SYSTEM temexdmod
  (* Version 1.0, Author, 4DIAC-Consortium *)
  APPLICATION looptest
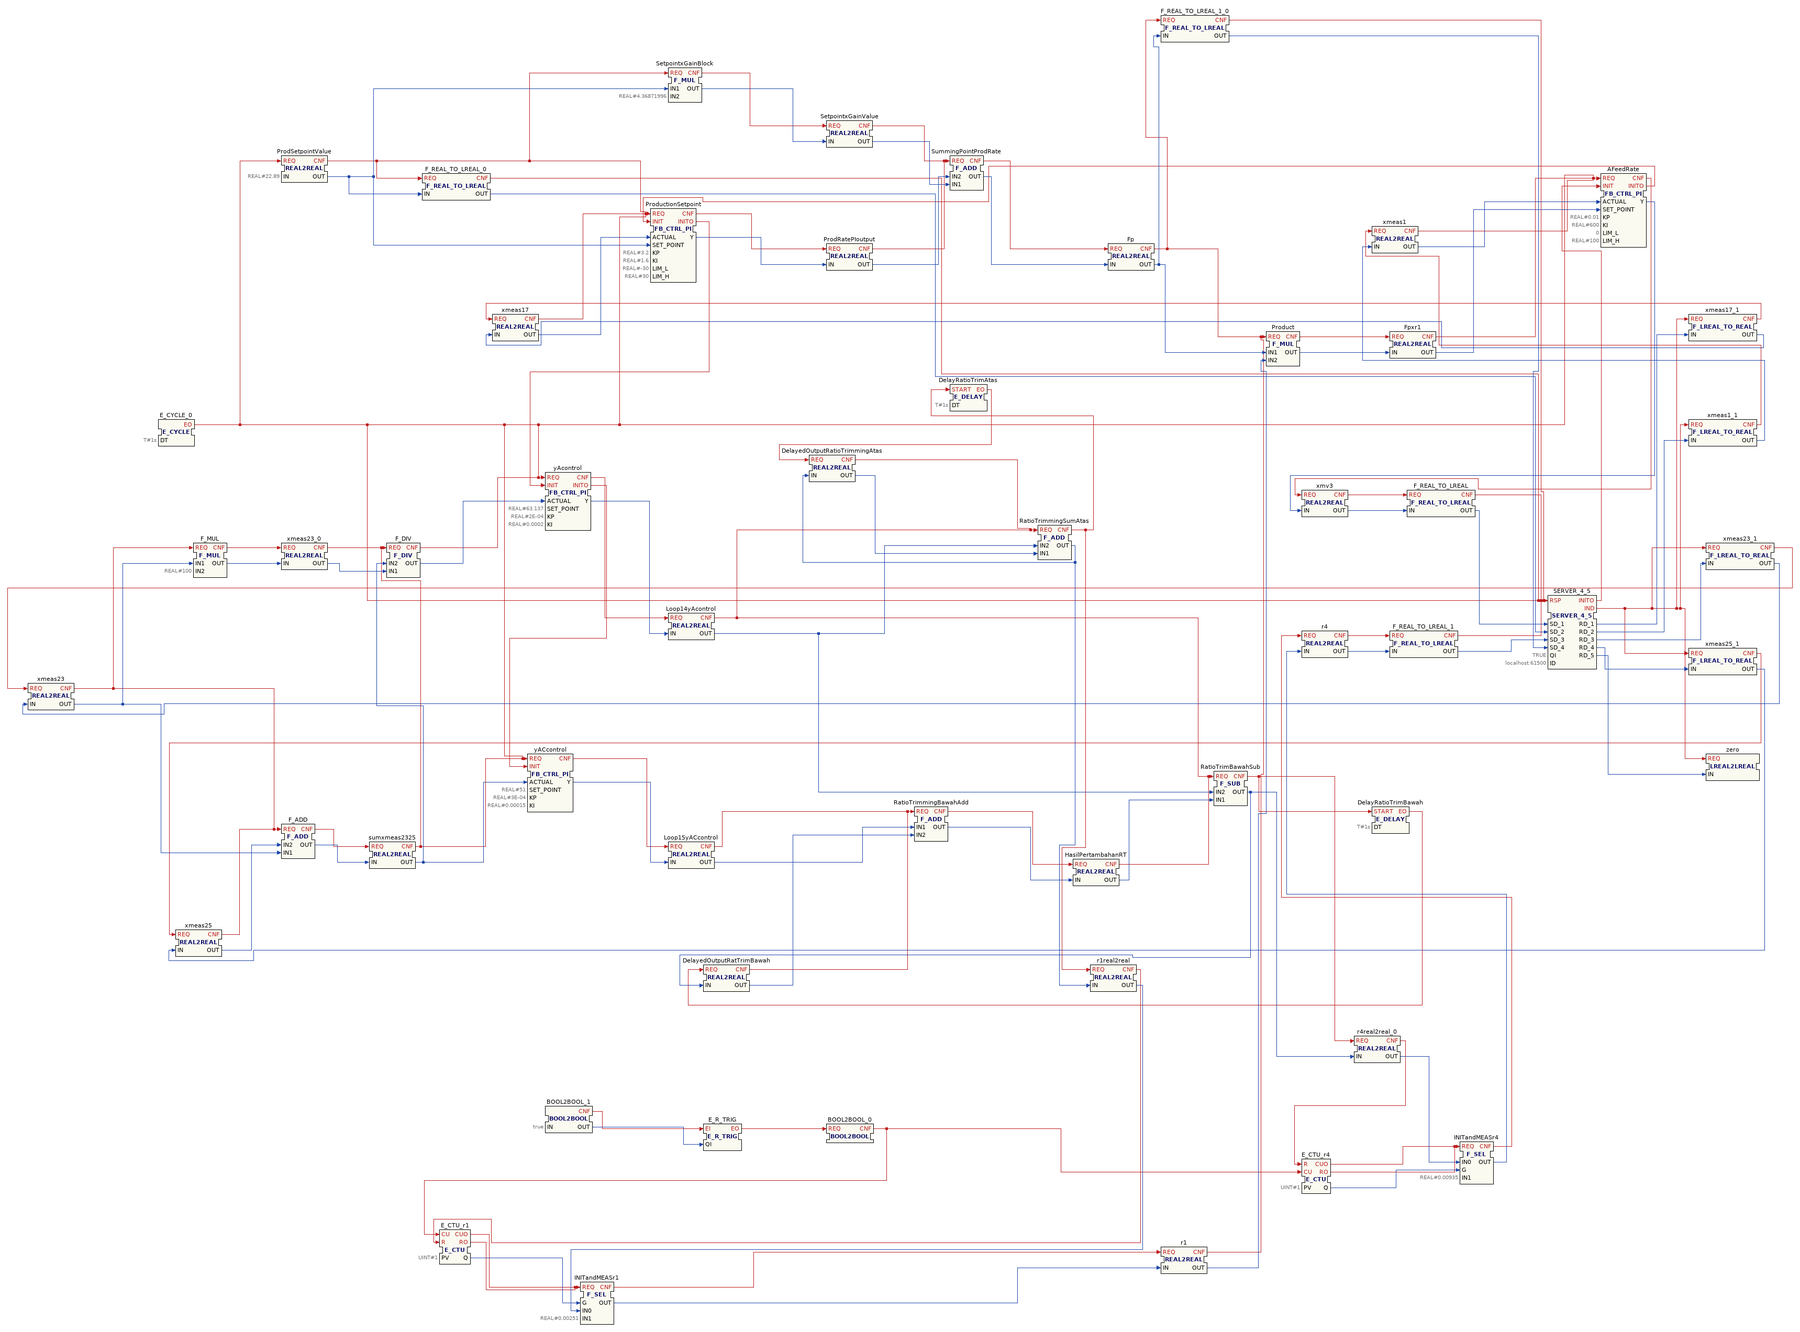
    FBS
      AFeedRate : FB_CTRL_PI(KP := REAL#0.01, KI := REAL#600, LIM_L := 0, LIM_H := REAL#100);
      ProductionSetpoint : FB_CTRL_PI(KP := REAL#3.2, KI := REAL#1.6, LIM_L := REAL#-30, LIM_H := REAL#30);
      Product : F_MUL;
      xmeas1 : REAL2REAL;
      Fpxr1 : REAL2REAL;
      xmv3 : REAL2REAL;
      SummingPointProdRate : F_ADD;
      ProdRatePIoutput : REAL2REAL;
      Fp : REAL2REAL;
      SetpointxGainBlock : F_MUL(IN2 := REAL#4.36871996);
      SetpointxGainValue : REAL2REAL;
      yAcontrol : FB_CTRL_PI(SET_POINT := REAL#63.137, KP := REAL#2E-04, KI := REAL#0.0002);
      yACcontrol : FB_CTRL_PI(SET_POINT := REAL#51, KP := REAL#3E-04, KI := REAL#0.00015);
      Loop14yAcontrol : REAL2REAL;
      Loop15yACcontrol : REAL2REAL;
      RatioTrimBawahSub : F_SUB;
      RatioTrimmingBawahAdd : F_ADD;
      HasilPertambahanRT : REAL2REAL;
      DelayRatioTrimBawah : E_DELAY(DT := T#1s);
      DelayedOutputRatTrimBawah : REAL2REAL;
      r4 : REAL2REAL;
      RatioTrimmingSumAtas : F_ADD;
      DelayedOutputRatioTrimmingAtas : REAL2REAL;
      DelayRatioTrimAtas : E_DELAY(DT := T#1s);
      xmeas17 : REAL2REAL;
      xmeas25 : REAL2REAL;
      F_ADD : F_ADD;
      sumxmeas2325 : REAL2REAL;
      F_MUL : F_MUL(IN2 := REAL#100);
      F_DIV : F_DIV;
      BOOL2BOOL_0 : BOOL2BOOL;
      E_CTU_r1 : E_CTU(PV := UINT#1);
      E_CYCLE_0 : E_CYCLE(DT := T#1s);
      r1real2real : REAL2REAL;
      BOOL2BOOL_1 : BOOL2BOOL(IN := true);
      INITandMEASr1 : F_SEL(IN1 := REAL#0.00251);
      E_R_TRIG : E_R_TRIG;
      r1 : REAL2REAL;
      SERVER_4_5 : SERVER_4_5(QI := TRUE, ID := localhost:61500);
      E_CTU_r4 : E_CTU(PV := UINT#1);
      INITandMEASr4 : F_SEL(IN1 := REAL#0.00935);
      r4real2real_0 : REAL2REAL;
      ProdSetpointValue : REAL2REAL(IN := REAL#22.89);
      F_REAL_TO_LREAL : F_REAL_TO_LREAL;
      F_REAL_TO_LREAL_0 : F_REAL_TO_LREAL;
      F_REAL_TO_LREAL_1 : F_REAL_TO_LREAL;
      F_REAL_TO_LREAL_1_0 : F_REAL_TO_LREAL;
      xmeas17_1 : F_LREAL_TO_REAL;
      xmeas1_1 : F_LREAL_TO_REAL;
      xmeas23_1 : F_LREAL_TO_REAL;
      xmeas25_1 : F_LREAL_TO_REAL;
      xmeas23 : REAL2REAL;
      xmeas23_0 : REAL2REAL;
      zero : LREAL2LREAL;
    END_FBS
    EVENT_CONNECTIONS
      Loop15yACcontrol.CNF TO RatioTrimmingBawahAdd.REQ;
      RatioTrimBawahSub.CNF TO DelayRatioTrimBawah.START;
      DelayRatioTrimBawah.EO TO DelayedOutputRatTrimBawah.REQ;
      DelayedOutputRatTrimBawah.CNF TO RatioTrimmingBawahAdd.REQ;
      Loop14yAcontrol.CNF TO RatioTrimmingSumAtas.REQ;
      Fp.CNF TO Product.REQ;
      RatioTrimmingSumAtas.CNF TO DelayRatioTrimAtas.START;
      DelayRatioTrimAtas.EO TO DelayedOutputRatioTrimmingAtas.REQ;
      DelayedOutputRatioTrimmingAtas.CNF TO RatioTrimmingSumAtas.REQ;
      SummingPointProdRate.CNF TO Fp.REQ;
      xmeas17.CNF TO ProductionSetpoint.REQ;
      SetpointxGainBlock.CNF TO SetpointxGainValue.REQ;
      SetpointxGainValue.CNF TO SummingPointProdRate.REQ;
      ProductionSetpoint.CNF TO ProdRatePIoutput.REQ;
      ProdRatePIoutput.CNF TO SummingPointProdRate.REQ;
      F_ADD.CNF TO sumxmeas2325.REQ;
      xmeas25.CNF TO F_ADD.REQ;
      sumxmeas2325.CNF TO yACcontrol.REQ;
      yACcontrol.CNF TO Loop15yACcontrol.REQ;
      F_DIV.CNF TO yAcontrol.REQ;
      yAcontrol.CNF TO Loop14yAcontrol.REQ;
      RatioTrimmingBawahAdd.CNF TO HasilPertambahanRT.REQ;
      HasilPertambahanRT.CNF TO RatioTrimBawahSub.REQ;
      Loop14yAcontrol.CNF TO RatioTrimBawahSub.REQ;
      Product.CNF TO Fpxr1.REQ;
      Fpxr1.CNF TO AFeedRate.REQ;
      xmeas1.CNF TO AFeedRate.REQ;
      AFeedRate.CNF TO xmv3.REQ;
      BOOL2BOOL_1.CNF TO E_R_TRIG.EI;
      E_R_TRIG.EO TO BOOL2BOOL_0.REQ;
      E_CTU_r1.CUO TO INITandMEASr1.REQ;
      E_CTU_r1.RO TO INITandMEASr1.REQ;
      BOOL2BOOL_0.CNF TO E_CTU_r1.CU;
      r1.CNF TO Product.REQ;
      RatioTrimmingSumAtas.CNF TO r1real2real.REQ;
      r1real2real.CNF TO E_CTU_r1.R;
      INITandMEASr1.CNF TO r1.REQ;
      AFeedRate.INITO TO ProductionSetpoint.INIT;
      ProductionSetpoint.INITO TO yAcontrol.INIT;
      yAcontrol.INITO TO yACcontrol.INIT;
      E_CYCLE_0.EO TO ProductionSetpoint.REQ;
      E_CYCLE_0.EO TO yAcontrol.REQ;
      E_CYCLE_0.EO TO yACcontrol.REQ;
      E_CYCLE_0.EO TO AFeedRate.REQ;
      SERVER_4_5.INITO TO AFeedRate.INIT;
      E_CYCLE_0.EO TO SERVER_4_5.RSP;
      INITandMEASr4.CNF TO r4.REQ;
      r4real2real_0.CNF TO E_CTU_r4.R;
      RatioTrimBawahSub.CNF TO r4real2real_0.REQ;
      BOOL2BOOL_0.CNF TO E_CTU_r4.CU;
      E_CTU_r4.CUO TO INITandMEASr4.REQ;
      E_CTU_r4.RO TO INITandMEASr4.REQ;
      E_CYCLE_0.EO TO ProdSetpointValue.REQ;
      ProdSetpointValue.CNF TO SetpointxGainBlock.REQ;
      ProdSetpointValue.CNF TO ProductionSetpoint.REQ;
      xmv3.CNF TO F_REAL_TO_LREAL.REQ;
      F_REAL_TO_LREAL.CNF TO SERVER_4_5.RSP;
      ProdSetpointValue.CNF TO F_REAL_TO_LREAL_0.REQ;
      F_REAL_TO_LREAL_0.CNF TO SERVER_4_5.RSP;
      r4.CNF TO F_REAL_TO_LREAL_1.REQ;
      F_REAL_TO_LREAL_1.CNF TO SERVER_4_5.RSP;
      F_REAL_TO_LREAL_1_0.CNF TO SERVER_4_5.RSP;
      Fp.CNF TO F_REAL_TO_LREAL_1_0.REQ;
      xmeas17_1.CNF TO xmeas17.REQ;
      SERVER_4_5.IND TO xmeas17_1.REQ;
      SERVER_4_5.IND TO xmeas1_1.REQ;
      xmeas1_1.CNF TO xmeas1.REQ;
      SERVER_4_5.IND TO xmeas23_1.REQ;
      xmeas23.CNF TO F_MUL.REQ;
      xmeas23.CNF TO F_ADD.REQ;
      xmeas23_1.CNF TO xmeas23.REQ;
      xmeas25_1.CNF TO xmeas25.REQ;
      SERVER_4_5.IND TO xmeas25_1.REQ;
      xmeas23_0.CNF TO F_DIV.REQ;
      F_MUL.CNF TO xmeas23_0.REQ;
      sumxmeas2325.CNF TO F_DIV.REQ;
      SERVER_4_5.IND TO zero.REQ;
    END_CONNECTIONS
    DATA_CONNECTIONS
      xmeas1.OUT TO AFeedRate.ACTUAL;
      Product.OUT TO Fpxr1.IN;
      Fpxr1.OUT TO AFeedRate.SET_POINT;
      AFeedRate.Y TO xmv3.IN;
      ProductionSetpoint.Y TO ProdRatePIoutput.IN;
      ProdRatePIoutput.OUT TO SummingPointProdRate.IN2;
      SummingPointProdRate.OUT TO Fp.IN;
      Fp.OUT TO Product.IN1;
      SetpointxGainBlock.OUT TO SetpointxGainValue.IN;
      SetpointxGainValue.OUT TO SummingPointProdRate.IN1;
      yAcontrol.Y TO Loop14yAcontrol.IN;
      yACcontrol.Y TO Loop15yACcontrol.IN;
      Loop14yAcontrol.OUT TO RatioTrimBawahSub.IN2;
      Loop15yACcontrol.OUT TO RatioTrimmingBawahAdd.IN1;
      RatioTrimmingBawahAdd.OUT TO HasilPertambahanRT.IN;
      HasilPertambahanRT.OUT TO RatioTrimBawahSub.IN1;
      RatioTrimBawahSub.OUT TO DelayedOutputRatTrimBawah.IN;
      DelayedOutputRatTrimBawah.OUT TO RatioTrimmingBawahAdd.IN2;
      Loop14yAcontrol.OUT TO RatioTrimmingSumAtas.IN2;
      RatioTrimmingSumAtas.OUT TO DelayedOutputRatioTrimmingAtas.IN;
      DelayedOutputRatioTrimmingAtas.OUT TO RatioTrimmingSumAtas.IN1;
      xmeas17.OUT TO ProductionSetpoint.ACTUAL;
      xmeas25.OUT TO F_ADD.IN2;
      F_ADD.OUT TO sumxmeas2325.IN;
      sumxmeas2325.OUT TO yACcontrol.ACTUAL;
      sumxmeas2325.OUT TO F_DIV.IN2;
      F_DIV.OUT TO yAcontrol.ACTUAL;
      E_CTU_r1.Q TO INITandMEASr1.G;
      BOOL2BOOL_1.OUT TO E_R_TRIG.QI;
      RatioTrimmingSumAtas.OUT TO r1real2real.IN;
      r1real2real.OUT TO INITandMEASr1.IN0;
      INITandMEASr1.OUT TO r1.IN;
      r1.OUT TO Product.IN2;
      INITandMEASr4.OUT TO r4.IN;
      RatioTrimBawahSub.OUT TO r4real2real_0.IN;
      r4real2real_0.OUT TO INITandMEASr4.IN0;
      E_CTU_r4.Q TO INITandMEASr4.G;
      ProdSetpointValue.OUT TO ProductionSetpoint.SET_POINT;
      ProdSetpointValue.OUT TO SetpointxGainBlock.IN1;
      xmv3.OUT TO F_REAL_TO_LREAL.IN;
      F_REAL_TO_LREAL.OUT TO SERVER_4_5.SD_1;
      ProdSetpointValue.OUT TO F_REAL_TO_LREAL_0.IN;
      F_REAL_TO_LREAL_0.OUT TO SERVER_4_5.SD_2;
      r4.OUT TO F_REAL_TO_LREAL_1.IN;
      F_REAL_TO_LREAL_1.OUT TO SERVER_4_5.SD_3;
      Fp.OUT TO F_REAL_TO_LREAL_1_0.IN;
      F_REAL_TO_LREAL_1_0.OUT TO SERVER_4_5.SD_4;
      xmeas17_1.OUT TO xmeas17.IN;
      SERVER_4_5.RD_1 TO xmeas17_1.IN;
      xmeas1_1.OUT TO xmeas1.IN;
      SERVER_4_5.RD_2 TO xmeas1_1.IN;
      SERVER_4_5.RD_3 TO xmeas23_1.IN;
      xmeas23.OUT TO F_ADD.IN1;
      xmeas23.OUT TO F_MUL.IN1;
      xmeas23_1.OUT TO xmeas23.IN;
      xmeas25_1.OUT TO xmeas25.IN;
      SERVER_4_5.RD_4 TO xmeas25_1.IN;
      xmeas23_0.OUT TO F_DIV.IN1;
      F_MUL.OUT TO xmeas23_0.IN;
      SERVER_4_5.RD_5 TO zero.IN;
    END_CONNECTIONS
  END_APPLICATION
  APPLICATION testfunctionblockbaru
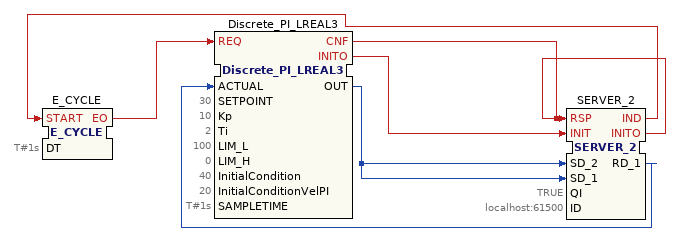
    FBS
      E_CYCLE : E_CYCLE(DT := T#1s);
      SERVER_2 : SERVER_2(QI := TRUE, ID := localhost:61500);
      Discrete_PI_LREAL3 : Discrete_PI_LREAL3(SETPOINT := 30, Kp := 10, Ti := 2, LIM_L := 100, LIM_H := 0, InitialCondition := 40, InitialConditionVelPI := 20, SAMPLETIME := T#1s);
    END_FBS
    EVENT_CONNECTIONS
      SERVER_2.IND TO E_CYCLE.START;
      SERVER_2.INITO TO SERVER_2.RSP;
      Discrete_PI_LREAL3.CNF TO SERVER_2.RSP;
      Discrete_PI_LREAL3.INITO TO SERVER_2.INIT;
      E_CYCLE.EO TO Discrete_PI_LREAL3.REQ;
    END_CONNECTIONS
    DATA_CONNECTIONS
      SERVER_2.RD_1 TO Discrete_PI_LREAL3.ACTUAL;
      Discrete_PI_LREAL3.OUT TO SERVER_2.SD_2;
      Discrete_PI_LREAL3.OUT TO SERVER_2.SD_1;
    END_CONNECTIONS
  END_APPLICATION
  APPLICATION tes
  END_APPLICATION
  APPLICATION testfunctionpid
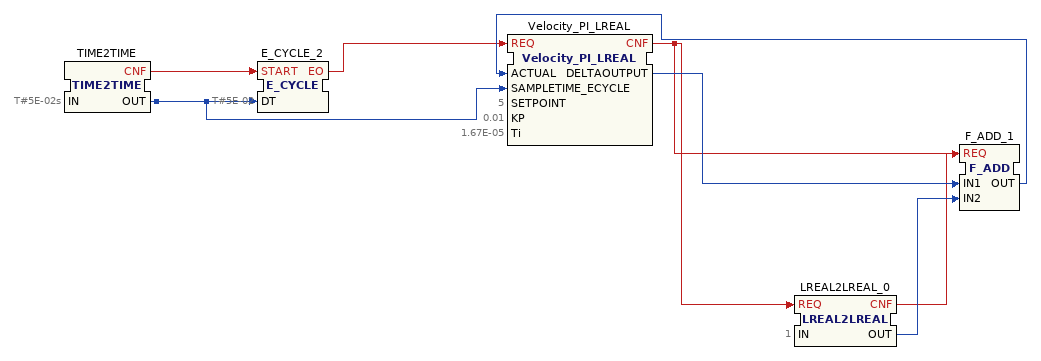
    FBS
      Velocity_PI_LREAL : Velocity_PI_LREAL(SETPOINT := 5, KP := 0.01, Ti := 1.67E-05);
      E_CYCLE_2 : E_CYCLE(DT := T#5E-02);
      F_ADD_1 : F_ADD;
      LREAL2LREAL_0 : LREAL2LREAL(IN := 1);
      TIME2TIME : TIME2TIME(IN := T#5E-02s);
    END_FBS
    EVENT_CONNECTIONS
      E_CYCLE_2.EO TO Velocity_PI_LREAL.REQ;
      Velocity_PI_LREAL.CNF TO F_ADD_1.REQ;
      Velocity_PI_LREAL.CNF TO LREAL2LREAL_0.REQ;
      LREAL2LREAL_0.CNF TO F_ADD_1.REQ;
      TIME2TIME.CNF TO E_CYCLE_2.START;
    END_CONNECTIONS
    DATA_CONNECTIONS
      Velocity_PI_LREAL.DELTAOUTPUT TO F_ADD_1.IN1;
      F_ADD_1.OUT TO Velocity_PI_LREAL.ACTUAL;
      LREAL2LREAL_0.OUT TO F_ADD_1.IN2;
      TIME2TIME.OUT TO E_CYCLE_2.DT;
      TIME2TIME.OUT TO Velocity_PI_LREAL.SAMPLETIME_ECYCLE;
    END_CONNECTIONS
  END_APPLICATION
  APPLICATION pressureloop2
    FBS
      xmeas17 : LREAL2LREAL;
      ProdRatePIDoutputLREAL_0 : LREAL2LREAL;
      K_0 : F_MUL;
      prodsetpointLREAL_0 : LREAL2LREAL(IN := 22.89);
      F_ADD_0_0 : F_ADD;
      F_MUL_0_0 : F_MUL;
      E_CYCLE_1_0 : E_CYCLE(DT := T#5E-02);
      xmeas7 : LREAL2LREAL;
      xmeas10 : LREAL2LREAL;
      SetpoxGain : LREAL2LREAL;
      Fp : LREAL2LREAL;
      r5 : LREAL2LREAL;
      NilaiK : LREAL2LREAL(IN := 4.3687);
      SERVER_3_5 : SERVER_3_5(QI := TRUE, ID := localhost:61500);
      PctGsp : LREAL2LREAL(IN := 53.8);
      xmv6 : LREAL2LREAL;
      PolymAtas : ADD_3(IN3 := 2.7690E-001);
      F_MUL_3 : F_MUL;
      FirstOrder : F_MUL(IN2 := 5.9446E-001);
      SecondOrder : F_MUL(IN2 := 1.5192E-003);
      Pangkat2 : LREAL2LREAL;
      HasilSecondOrder : LREAL2LREAL;
      HasilFirstOrder : LREAL2LREAL;
      SecondOrder_0 : F_MUL(IN2 := -1.1377E-003);
      HasilSecondOrder_0 : LREAL2LREAL;
      FirstOrder_0 : F_MUL(IN2 := -8.0893E-001);
      HasilFirstOrder_0 : LREAL2LREAL;
      PolymBawah : ADD_3(IN3 := 9.1060E+001);
      F_MUL_7 : F_MUL(IN2 := 32);
      F_MUL_8 : F_MUL(IN2 := 46);
      LREAL2LREAL_10 : LREAL2LREAL;
      LREAL2LREAL_11 : LREAL2LREAL;
      F_DIV_0 : F_DIV;
      LREAL2LREAL_12 : LREAL2LREAL;
      LREAL2LREAL_13 : LREAL2LREAL;
      r3 : F_ADD;
      r2 : F_SUB;
      LREAL2LREAL_14 : LREAL2LREAL;
      F_DIV_1 : F_DIV;
      LREAL2LREAL_15 : LREAL2LREAL;
      r3_1 : LREAL2LREAL;
      F_MUL_9 : F_MUL;
      xmeas40 : LREAL2LREAL;
      xmeas3 : LREAL2LREAL;
      xmv2 : LREAL2LREAL;
      ProductionRate : Discrete_PI_LREAL2(Kp := 3.2, Ti := 2, LIM_L := 30, LIM_H := 30, InitialCondition := -0.4489, InitialConditionVelPI := -0.1407, SAMPLETIME := T#50ms);
      ReactorPressure : Discrete_PI_LREAL2(SETPOINT := 2800, Kp := -1E-04, Ti := 0.333, LIM_L := 0, LIM_H := 100, InitialCondition := 0.0019, InitialConditionVelPI := 1.0409, SAMPLETIME := T#50ms);
      PurgeRate : Discrete_PI_LREAL2(Kp := 0.01, Ti := 167E-05, LIM_L := 0, LIM_H := 100, InitialCondition := 24.2293, InitialConditionVelPI := -0.0064, SAMPLETIME := T#50ms);
      GinProduct : Discrete_PI_LREAL2(Kp := -0.4, Ti := 1.6667, LIM_L := -inf, LIM_H := inf, InitialCondition := 0.6323, InitialConditionVelPI := -0.5067, SAMPLETIME := T#50ms);
      EFeedRate : Discrete_PI_LREAL2(Kp := 1.8E-6, Ti := 1.667E-05, LIM_L := 0, LIM_H := 100, InitialCondition := 53.3867, InitialConditionVelPI := 9.7234, SAMPLETIME := T#50ms);
      TIME2TIME_0 : TIME2TIME(IN := T#1ms);
      LREAL2LREAL_3 : LREAL2LREAL(IN := 2.7690E-001);
      LREAL2LREAL_3_0 : LREAL2LREAL(IN := 5.9446E-001);
      LREAL2LREAL_5 : LREAL2LREAL(IN := -1.1377E-003);
      LREAL2LREAL_6 : LREAL2LREAL(IN := -8.0893E-001);
      LREAL2LREAL_4 : LREAL2LREAL(IN := 9.1060E+001);
      LREAL2LREAL_7 : LREAL2LREAL(IN := 32);
      LREAL2LREAL_8 : LREAL2LREAL(IN := 46);
      LREAL2LREAL_9 : LREAL2LREAL(IN := 1.5192E-003);
      r2_1 : LREAL2LREAL;
      F_MUL_10 : F_MUL;
      DFeedRate : Discrete_PI_LREAL2(Kp := 1.6E-6, Ti := 1.667E-05, LIM_L := 0, LIM_H := 100, InitialCondition := 53.3867, InitialConditionVelPI := 9.7234);
      xmv1 : LREAL2LREAL;
      xmeas2 : LREAL2LREAL;
      SERVER_3_5_0 : SERVER_3_5(QI := TRUE, ID := localhost:61501);
      xmeas23 : LREAL2LREAL;
      xmeas25 : LREAL2LREAL;
      F_ADD_0 : F_ADD;
      F_MUL_0 : F_MUL;
      F_DIV_2 : F_DIV;
      Gain100 : LREAL2LREAL(IN := 100);
      yAC : LREAL2LREAL(IN := 100);
      yA : LREAL2LREAL(IN := 100);
      xmeas23x100 : LREAL2LREAL(IN := 100);
      yAcontrolLoop14 : Velocity_PI_LREAL2(KP := 2E-4, Ti := 1, InitialCondition := 0.1568, SAMPLETIME_ECYCLE := 100ms);
      yACcontrolLoop15 : Velocity_PI_LREAL2(KP := 3E-4, Ti := 2, InitialCondition := -0.1936, SAMPLETIME_ECYCLE := 100ms);
      F_ADD_2 : F_ADD;
      F_ADD_3 : F_ADD;
      F_SUB : F_SUB;
      Delay_With_InitCondition : Delay_With_InitCondition(DelayTime := 100ms, InitialCondition := 0.002722836244293);
      Delay_With_InitCondition_0 : Delay_With_InitCondition(DelayTime := 100ms, InitialCondition := 0.092236609900323);
      summmingpoinloop15 : LREAL2LREAL;
      r1 : LREAL2LREAL;
      r4 : LREAL2LREAL;
      AFeedRate : Discrete_PI_LREAL2;
      CFeedRate : Discrete_PI_LREAL2;
      r1xFp : F_MUL;
      r4xFp : F_MUL;
      xmeas1 : LREAL2LREAL;
      xmeas4 : LREAL2LREAL;
      xmv3 : LREAL2LREAL;
      xmv4 : LREAL2LREAL;
    END_FBS
    EVENT_CONNECTIONS
      ProdRatePIDoutputLREAL_0.CNF TO F_ADD_0_0.REQ;
      SetpoxGain.CNF TO F_ADD_0_0.REQ;
      K_0.CNF TO SetpoxGain.REQ;
      F_ADD_0_0.CNF TO Fp.REQ;
      NilaiK.CNF TO K_0.REQ;
      r5.CNF TO F_MUL_0_0.REQ;
      Fp.CNF TO F_MUL_0_0.REQ;
      PctGsp.CNF TO F_MUL_3.REQ;
      F_MUL_3.CNF TO Pangkat2.REQ;
      Pangkat2.CNF TO SecondOrder.REQ;
      PctGsp.CNF TO FirstOrder.REQ;
      SecondOrder.CNF TO HasilSecondOrder.REQ;
      HasilSecondOrder.CNF TO PolymAtas.REQ;
      FirstOrder.CNF TO HasilFirstOrder.REQ;
      HasilFirstOrder.CNF TO PolymAtas.REQ;
      Pangkat2.CNF TO SecondOrder_0.REQ;
      FirstOrder_0.CNF TO HasilFirstOrder_0.REQ;
      SecondOrder_0.CNF TO HasilSecondOrder_0.REQ;
      HasilSecondOrder_0.CNF TO PolymBawah.REQ;
      HasilFirstOrder_0.CNF TO PolymBawah.REQ;
      F_MUL_8.CNF TO LREAL2LREAL_10.REQ;
      F_MUL_7.CNF TO LREAL2LREAL_11.REQ;
      PolymBawah.CNF TO LREAL2LREAL_12.REQ;
      LREAL2LREAL_10.CNF TO F_DIV_0.REQ;
      F_DIV_0.CNF TO LREAL2LREAL_14.REQ;
      LREAL2LREAL_14.CNF TO r3.REQ;
      LREAL2LREAL_12.CNF TO r3.REQ;
      PolymAtas.CNF TO LREAL2LREAL_13.REQ;
      LREAL2LREAL_13.CNF TO r2.REQ;
      LREAL2LREAL_11.CNF TO F_DIV_1.REQ;
      F_DIV_1.CNF TO LREAL2LREAL_15.REQ;
      LREAL2LREAL_15.CNF TO r2.REQ;
      r3.CNF TO r3_1.REQ;
      r3_1.CNF TO F_MUL_9.REQ;
      SERVER_3_5.INITO TO ProductionRate.INIT;
      xmeas17.CNF TO ProductionRate.REQ;
      prodsetpointLREAL_0.CNF TO ProductionRate.REQ;
      ProductionRate.CNF TO K_0.REQ;
      ProductionRate.CNF TO ProdRatePIDoutputLREAL_0.REQ;
      ProductionRate.INITO TO ReactorPressure.INIT;
      xmeas7.CNF TO ReactorPressure.REQ;
      ReactorPressure.CNF TO r5.REQ;
      ReactorPressure.INITO TO PurgeRate.INIT;
      xmeas10.CNF TO PurgeRate.REQ;
      F_MUL_0_0.CNF TO PurgeRate.REQ;
      PurgeRate.CNF TO xmv6.REQ;
      PurgeRate.INITO TO GinProduct.INIT;
      xmeas40.CNF TO GinProduct.REQ;
      PctGsp.CNF TO GinProduct.REQ;
      GinProduct.CNF TO F_MUL_7.REQ;
      GinProduct.CNF TO F_MUL_8.REQ;
      GinProduct.INITO TO EFeedRate.INIT;
      F_MUL_9.CNF TO EFeedRate.REQ;
      EFeedRate.CNF TO xmv2.REQ;
      ProductionRate.CNF TO NilaiK.REQ;
      LREAL2LREAL_3.CNF TO PolymAtas.REQ;
      HasilFirstOrder.CNF TO LREAL2LREAL_3.REQ;
      PctGsp.CNF TO LREAL2LREAL_3_0.REQ;
      Pangkat2.CNF TO LREAL2LREAL_5.REQ;
      LREAL2LREAL_6.CNF TO FirstOrder_0.REQ;
      PctGsp.CNF TO LREAL2LREAL_6.REQ;
      LREAL2LREAL_4.CNF TO PolymBawah.REQ;
      HasilSecondOrder_0.CNF TO LREAL2LREAL_4.REQ;
      LREAL2LREAL_7.CNF TO F_MUL_7.REQ;
      GinProduct.CNF TO LREAL2LREAL_7.REQ;
      LREAL2LREAL_8.CNF TO F_MUL_8.REQ;
      GinProduct.CNF TO LREAL2LREAL_8.REQ;
      LREAL2LREAL_9.CNF TO SecondOrder.REQ;
      Pangkat2.CNF TO LREAL2LREAL_9.REQ;
      SERVER_3_5.IND TO xmeas10.REQ;
      SERVER_3_5.IND TO xmeas7.REQ;
      SERVER_3_5.IND TO PctGsp.REQ;
      SERVER_3_5.IND TO xmeas40.REQ;
      SERVER_3_5.IND TO xmeas3.REQ;
      SERVER_3_5.IND TO xmeas17.REQ;
      SERVER_3_5.IND TO prodsetpointLREAL_0.REQ;
      xmv2.CNF TO E_CYCLE_1_0.START;
      TIME2TIME_0.CNF TO E_CYCLE_1_0.START;
      xmv6.CNF TO E_CYCLE_1_0.START;
      E_CYCLE_1_0.EO TO SERVER_3_5.RSP;
      r2.CNF TO r2_1.REQ;
      r2_1.CNF TO F_MUL_10.REQ;
      F_MUL_10.CNF TO DFeedRate.REQ;
      xmeas3.CNF TO EFeedRate.REQ;
      xmeas2.CNF TO DFeedRate.REQ;
      DFeedRate.CNF TO xmv1.REQ;
      xmv1.CNF TO E_CYCLE_1_0.START;
      Fp.CNF TO F_MUL_9.REQ;
      Fp.CNF TO F_MUL_10.REQ;
      Fp.CNF TO F_DIV_1.REQ;
      Fp.CNF TO F_DIV_0.REQ;
      SERVER_3_5_0.INITO TO DFeedRate.INIT;
      SERVER_3_5_0.IND TO xmeas2.REQ;
      E_CYCLE_1_0.EO TO SERVER_3_5_0.RSP;
      SERVER_3_5_0.IND TO xmeas23.REQ;
      SERVER_3_5_0.IND TO xmeas25.REQ;
      Gain100.CNF TO F_MUL_0.REQ;
      xmeas23.CNF TO Gain100.REQ;
      xmeas25.CNF TO F_ADD_0.REQ;
      F_ADD_0.CNF TO yAC.REQ;
      F_MUL_0.CNF TO xmeas23x100.REQ;
      xmeas23x100.CNF TO F_DIV_2.REQ;
      F_DIV_2.CNF TO yA.REQ;
      DFeedRate.INITO TO yACcontrolLoop15.INIT;
      yACcontrolLoop15.INITO TO yAcontrolLoop14.INIT;
      yA.CNF TO yAcontrolLoop14.REQ;
      yAC.CNF TO yACcontrolLoop15.REQ;
      yAcontrolLoop14.INITO TO Delay_With_InitCondition.INIT;
      yAcontrolLoop14.CNF TO F_ADD_2.REQ;
      F_ADD_2.CNF TO Delay_With_InitCondition.Start_and_REQ;
      yACcontrolLoop15.CNF TO F_ADD_3.REQ;
      yACcontrolLoop15.INITO TO Delay_With_InitCondition_0.INIT;
      F_ADD_3.CNF TO summmingpoinloop15.REQ;
      summmingpoinloop15.CNF TO F_SUB.REQ;
      F_SUB.CNF TO Delay_With_InitCondition_0.Start_and_REQ;
      F_ADD_2.CNF TO r1.REQ;
      F_SUB.CNF TO r4.REQ;
      Delay_With_InitCondition.CNF TO F_ADD_2.REQ;
      Delay_With_InitCondition_0.CNF TO F_ADD_3.REQ;
      yAcontrolLoop14.INITO TO AFeedRate.INIT;
      AFeedRate.INITO TO CFeedRate.INIT;
      r1.CNF TO r1xFp.REQ;
      r4.CNF TO r4xFp.REQ;
      Fp.CNF TO r1xFp.REQ;
      Fp.CNF TO r4xFp.REQ;
      r1xFp.CNF TO AFeedRate.REQ;
      r4xFp.CNF TO CFeedRate.REQ;
      SERVER_3_5_0.IND TO xmeas1.REQ;
      SERVER_3_5_0.IND TO xmeas4.REQ;
      xmeas1.CNF TO AFeedRate.REQ;
      xmeas4.CNF TO CFeedRate.REQ;
      xmv4.CNF TO E_CYCLE_1_0.START;
      xmv3.CNF TO E_CYCLE_1_0.START;
      AFeedRate.CNF TO xmv3.REQ;
      CFeedRate.CNF TO xmv4.REQ;
      LREAL2LREAL_3_0.CNF TO FirstOrder.REQ;
      LREAL2LREAL_5.CNF TO SecondOrder_0.REQ;
    END_CONNECTIONS
    DATA_CONNECTIONS
      ProdRatePIDoutputLREAL_0.OUT TO F_ADD_0_0.IN2;
      SetpoxGain.OUT TO F_ADD_0_0.IN1;
      K_0.OUT TO SetpoxGain.IN;
      F_ADD_0_0.OUT TO Fp.IN;
      ProdRatePIDoutputLREAL_0.OUT TO K_0.IN1;
      NilaiK.OUT TO K_0.IN2;
      r5.OUT TO F_MUL_0_0.IN2;
      Fp.OUT TO F_MUL_0_0.IN1;
      SERVER_3_5.RD_1 TO xmeas17.IN;
      SERVER_3_5.RD_2 TO xmeas7.IN;
      SERVER_3_5.RD_3 TO xmeas10.IN;
      xmv6.OUT TO SERVER_3_5.SD_1;
      PctGsp.OUT TO F_MUL_3.IN1;
      PctGsp.OUT TO F_MUL_3.IN2;
      F_MUL_3.OUT TO Pangkat2.IN;
      Pangkat2.OUT TO SecondOrder.IN1;
      PctGsp.OUT TO FirstOrder.IN1;
      SecondOrder.OUT TO HasilSecondOrder.IN;
      HasilSecondOrder.OUT TO PolymAtas.IN1;
      FirstOrder.OUT TO HasilFirstOrder.IN;
      HasilFirstOrder.OUT TO PolymAtas.IN2;
      Pangkat2.OUT TO SecondOrder_0.IN1;
      PctGsp.OUT TO FirstOrder_0.IN1;
      FirstOrder_0.OUT TO HasilFirstOrder_0.IN;
      SecondOrder_0.OUT TO HasilSecondOrder_0.IN;
      HasilSecondOrder_0.OUT TO PolymBawah.IN1;
      HasilFirstOrder_0.OUT TO PolymBawah.IN2;
      F_MUL_8.OUT TO LREAL2LREAL_10.IN;
      F_MUL_7.OUT TO LREAL2LREAL_11.IN;
      LREAL2LREAL_10.OUT TO F_DIV_0.IN1;
      PolymBawah.OUT TO LREAL2LREAL_12.IN;
      F_DIV_0.OUT TO LREAL2LREAL_14.IN;
      LREAL2LREAL_14.OUT TO r3.IN1;
      LREAL2LREAL_12.OUT TO r3.IN2;
      PolymAtas.OUT TO LREAL2LREAL_13.IN;
      LREAL2LREAL_13.OUT TO r2.IN1;
      LREAL2LREAL_11.OUT TO F_DIV_1.IN1;
      F_DIV_1.OUT TO LREAL2LREAL_15.IN;
      LREAL2LREAL_15.OUT TO r2.IN2;
      r3.OUT TO r3_1.IN;
      r3_1.OUT TO F_MUL_9.IN1;
      SERVER_3_5.RD_4 TO xmeas40.IN;
      SERVER_3_5.RD_5 TO xmeas3.IN;
      xmv6.OUT TO SERVER_3_5.SD_2;
      xmv2.OUT TO SERVER_3_5.SD_3;
      xmeas17.OUT TO ProductionRate.ACTUAL;
      prodsetpointLREAL_0.OUT TO ProductionRate.SETPOINT;
      ProductionRate.OUT TO ProdRatePIDoutputLREAL_0.IN;
      xmeas7.OUT TO ReactorPressure.ACTUAL;
      ReactorPressure.OUT TO r5.IN;
      PurgeRate.OUT TO xmv6.IN;
      xmeas10.OUT TO PurgeRate.ACTUAL;
      F_MUL_0_0.OUT TO PurgeRate.SETPOINT;
      xmeas40.OUT TO GinProduct.ACTUAL;
      PctGsp.OUT TO GinProduct.SETPOINT;
      GinProduct.OUT TO F_MUL_8.IN1;
      GinProduct.OUT TO F_MUL_7.IN1;
      EFeedRate.OUT TO xmv2.IN;
      F_MUL_9.OUT TO EFeedRate.SETPOINT;
      xmeas3.OUT TO EFeedRate.ACTUAL;
      TIME2TIME_0.OUT TO ProductionRate.SAMPLETIME;
      TIME2TIME_0.OUT TO ReactorPressure.SAMPLETIME;
      TIME2TIME_0.OUT TO PurgeRate.SAMPLETIME;
      TIME2TIME_0.OUT TO GinProduct.SAMPLETIME;
      TIME2TIME_0.OUT TO EFeedRate.SAMPLETIME;
      LREAL2LREAL_3.OUT TO PolymAtas.IN3;
      LREAL2LREAL_3_0.OUT TO FirstOrder.IN2;
      LREAL2LREAL_5.OUT TO SecondOrder_0.IN2;
      LREAL2LREAL_6.OUT TO FirstOrder_0.IN2;
      LREAL2LREAL_4.OUT TO PolymBawah.IN3;
      LREAL2LREAL_7.OUT TO F_MUL_7.IN2;
      LREAL2LREAL_8.OUT TO F_MUL_8.IN2;
      LREAL2LREAL_9.OUT TO SecondOrder.IN2;
      TIME2TIME_0.OUT TO E_CYCLE_1_0.DT;
      r2.OUT TO r2_1.IN;
      r2_1.OUT TO F_MUL_10.IN1;
      F_MUL_10.OUT TO DFeedRate.SETPOINT;
      xmeas2.OUT TO DFeedRate.ACTUAL;
      DFeedRate.OUT TO xmv1.IN;
      TIME2TIME_0.OUT TO DFeedRate.SAMPLETIME;
      Fp.OUT TO F_MUL_9.IN2;
      Fp.OUT TO F_MUL_10.IN2;
      Fp.OUT TO F_DIV_1.IN2;
      Fp.OUT TO F_DIV_0.IN2;
      SERVER_3_5_0.RD_1 TO xmeas2.IN;
      xmv1.OUT TO SERVER_3_5_0.SD_1;
      SERVER_3_5_0.RD_2 TO xmeas23.IN;
      SERVER_3_5_0.RD_3 TO xmeas25.IN;
      xmeas23.OUT TO F_MUL_0.IN1;
      Gain100.OUT TO F_MUL_0.IN2;
      xmeas25.OUT TO F_ADD_0.IN2;
      xmeas23.OUT TO F_ADD_0.IN1;
      F_ADD_0.OUT TO yAC.IN;
      yAC.OUT TO F_DIV_2.IN2;
      F_MUL_0.OUT TO xmeas23x100.IN;
      xmeas23x100.OUT TO F_DIV_2.IN1;
      F_DIV_2.OUT TO yA.IN;
      yA.OUT TO yAcontrolLoop14.ACTUAL;
      yAC.OUT TO yACcontrolLoop15.ACTUAL;
      yAcontrolLoop14.DELTAOUTPUT TO F_ADD_2.IN1;
      Delay_With_InitCondition.LREAL1 TO F_ADD_2.IN2;
      F_ADD_2.OUT TO Delay_With_InitCondition.DelayedInput;
      yAcontrolLoop14.DELTAOUTPUT TO F_SUB.IN2;
      yACcontrolLoop15.DELTAOUTPUT TO F_ADD_3.IN1;
      Delay_With_InitCondition_0.LREAL1 TO F_ADD_3.IN2;
      F_ADD_3.OUT TO summmingpoinloop15.IN;
      summmingpoinloop15.OUT TO F_SUB.IN1;
      F_ADD_2.OUT TO r1.IN;
      F_SUB.OUT TO r4.IN;
      F_SUB.OUT TO Delay_With_InitCondition_0.DelayedInput;
      r1.OUT TO r1xFp.IN1;
      r4.OUT TO r4xFp.IN1;
      Fp.OUT TO r1xFp.IN2;
      Fp.OUT TO r4xFp.IN2;
      r1xFp.OUT TO AFeedRate.SETPOINT;
      r4xFp.OUT TO CFeedRate.SETPOINT;
      SERVER_3_5_0.RD_4 TO xmeas1.IN;
      SERVER_3_5_0.RD_5 TO xmeas4.IN;
      xmeas1.OUT TO AFeedRate.ACTUAL;
      xmeas4.OUT TO CFeedRate.ACTUAL;
      xmv4.OUT TO SERVER_3_5_0.SD_3;
      xmv3.OUT TO SERVER_3_5_0.SD_2;
      AFeedRate.OUT TO xmv3.IN;
      CFeedRate.OUT TO xmv4.IN;
    END_CONNECTIONS
  END_APPLICATION
  APPLICATION mode1
    FBS
      xmeas17 : LREAL2LREAL;
      ProdRatePIDoutputLREAL_0_0 : LREAL2LREAL;
      K_0_0 : F_MUL;
      prodsetpointLREAL_0_0 : LREAL2LREAL(IN := 22.89);
      F_ADD_0_0_0 : F_ADD;
      F_MUL_0_0_0 : F_MUL;
      E_CYCLE_1_0_0 : E_CYCLE;
      xmeas7 : LREAL2LREAL;
      xmeas10 : LREAL2LREAL;
      SetpoxGain_0 : LREAL2LREAL;
      Fp_0 : LREAL2LREAL;
      r5_0 : LREAL2LREAL;
      NilaiK_0 : LREAL2LREAL(IN := 4.3687);
      Server2 : SERVER_3_5(QI := TRUE, ID := localhost:61001);
      PctGsp_0 : LREAL2LREAL(IN := 53.8);
      xmv6_0 : LREAL2LREAL;
      r3_1_0 : LREAL2LREAL;
      F_MUL_9_0 : F_MUL;
      xmeas40 : LREAL2LREAL;
      xmeas3 : LREAL2LREAL;
      xmv2_0 : LREAL2LREAL;
      ProductionRate_0 : Discrete_PI_LREAL2(Kp := 3.2, Ti := 2, LIM_L := -30, LIM_H := 30, InitialCondition := -0.4489, InitialConditionVelPI := -0.1407);
      ReactorPressure_0 : Discrete_PI_LREAL2(SETPOINT := 2800, Kp := -1E-04, Ti := 0.333, LIM_L := 0, LIM_H := 100, InitialCondition := 0.0019, InitialConditionVelPI := 1.0409);
      PurgeRate_0 : Discrete_PI_LREAL2(Kp := 0.01, Ti := 167E-05, LIM_L := 0, LIM_H := 100, InitialCondition := 24.2293, InitialConditionVelPI := -0.0064);
      GinProduct_0 : Discrete_PI_LREAL2(Kp := -0.4, Ti := 1.6667, LIM_L := -inf, LIM_H := inf, InitialCondition := 0.6323, InitialConditionVelPI := -0.5067);
      EFeedRate_0 : Discrete_PI_LREAL2(Kp := 1.8E-6, Ti := 1.667E-05, LIM_L := 0, LIM_H := 100, InitialCondition := 53.3867, InitialConditionVelPI := 9.7234);
      TIME2TIME_0_0 : TIME2TIME(IN := T#1ms);
      r2_1_0 : LREAL2LREAL;
      F_MUL_10_0 : F_MUL;
      DFeedRate_0 : Discrete_PI_LREAL2(Kp := 1.6E-6, Ti := 1.667E-05, LIM_L := 0, LIM_H := 100, InitialCondition := 53.3867, InitialConditionVelPI := 9.7234);
      xmv1_0 : LREAL2LREAL;
      Server1 : SERVER_3_5(QI := TRUE, ID := localhost:61000);
      xmeas23 : LREAL2LREAL;
      xmeas25 : LREAL2LREAL;
      F_ADD_0_1 : F_ADD;
      F_MUL_0_1 : F_MUL;
      F_DIV_2_0 : F_DIV;
      Gain100_0 : LREAL2LREAL(IN := 100);
      yAC_0 : LREAL2LREAL;
      yA_0 : LREAL2LREAL;
      xmeas23x100_0 : LREAL2LREAL;
      yAcontrolLoop14_0 : Velocity_PI_LREAL2(SETPOINT := 63.13725, KP := 2E-4, Ti := 1, InitialCondition := 0.1568, SAMPLETIME_ECYCLE := T#100ms);
      yACcontrolLoop15_0 : Velocity_PI_LREAL2(SETPOINT := 51, KP := 3E-4, Ti := 2, InitialCondition := -0.1936, SAMPLETIME_ECYCLE := T#100ms);
      F_ADD_2_0 : F_ADD;
      F_ADD_3_0 : F_ADD;
      F_SUB_2 : F_SUB;
      Delay_With_InitCondition_1 : Delay_With_InitCondition(DelayTime := T#100ms, InitialCondition := 0.002722836244293);
      Delay_With_InitCondition_0_0 : Delay_With_InitCondition(DelayTime := T#100ms, InitialCondition := 0.092236609900323);
      summmingpoinloop15_0 : LREAL2LREAL;
      r1_0 : LREAL2LREAL;
      r4_0 : LREAL2LREAL;
      AFeedRate_0 : Discrete_PI_LREAL2(Kp := 0.01, Ti := 1.66667E-05, LIM_L := 0, LIM_H := 100, InitialCondition := 26.6622, InitialConditionVelPI := 0.0027);
      CFeedRate_0 : Discrete_PI_LREAL2(Kp := 0.003, Ti := 1.66667E-05, LIM_L := 0, LIM_H := 100, InitialCondition := 60.4829, InitialConditionVelPI := 0.0835);
      r1xFp_0 : F_MUL;
      r4xFp_0 : F_MUL;
      xmeas4 : LREAL2LREAL;
      xmv3_0 : LREAL2LREAL;
      xmv4_0 : LREAL2LREAL;
      Feedforward : Feedforward;
      xmeas12 : LREAL2LREAL;
      xmeas14 : LREAL2LREAL;
      SeparatorLevel : Discrete_PI_LREAL2(SETPOINT := 50, Kp := -0.001, Ti := 3.333333333, LIM_L := 0, LIM_H := 100, InitialCondition := 0.2537, InitialConditionVelPI := -1.0418);
      r6 : LREAL2LREAL;
      Fp : LREAL2LREAL;
      F_MUL_1 : F_MUL;
      SeparatorFlowRate : Discrete_PI_LREAL2(Kp := 0.0004, Ti := 1.66667E-05, LIM_L := 0, LIM_H := 100, InitialCondition := 37.2082, InitialConditionVelPI := 0.0481);
      xmv7 : LREAL2LREAL;
      xmeas15 : LREAL2LREAL;
      StripperLevel : Discrete_PI_LREAL2(SETPOINT := 50, Kp := -0.0002, Ti := 3.333333333, LIM_L := 0, LIM_H := 100, InitialCondition := 0.2287, InitialConditionVelPI := 0.9492);
      r7 : LREAL2LREAL;
      F_MUL_1_0 : F_MUL;
      StripperFlowRate : Discrete_PI_LREAL2(Kp := 0.0004, Ti := 1.66667E-05, LIM_L := 0, LIM_H := 100, InitialCondition := 37.2082, InitialConditionVelPI := 0.0481);
      xmv8 : LREAL2LREAL;
      xmeas11 : LREAL2LREAL;
      xmeas8 : LREAL2LREAL;
      xmeas9 : LREAL2LREAL;
      xmv10 : LREAL2LREAL;
      ReactorLevel : Discrete_PI_LREAL2(SETPOINT := 65, Kp := 0.8, Ti := 1, LIM_L := 0, LIM_H := 120, InitialCondition := 92.02, InitialConditionVelPI := 0.0408);
      ReactorTemperature : Discrete_PI_LREAL2(SETPOINT := 122.9, Kp := -8, Ti := 0.125, LIM_L := 0, LIM_H := 100, InitialCondition := 35.8653, InitialConditionVelPI := 0.008);
      SeparatorTemperature : Discrete_PI_LREAL2(Kp := -4, Ti := 0.25, LIM_L := 0, LIM_H := 100, InitialCondition := 12.9306, InitialConditionVelPI := -0.1416);
      xmv11 : LREAL2LREAL;
      Server3 : SERVER_3_5(QI := TRUE, ID := localhost:61002);
      Server4 : SERVER_4_2(QI := TRUE, ID := localhost:61003);
      xmv5 : LREAL2LREAL(IN := 0);
      xmv9 : LREAL2LREAL(IN := 0);
      xmv12 : LREAL2LREAL(IN := 100);
      xmeas17_2 : LREAL2LREAL;
      xmeas17_2_0 : LREAL2LREAL;
      RectorPressure_0 : FB_CTRL_PI;
      SeparatorLeel_0 : FB_CTRL_PI;
      StripperLevel_0 : FB_CTRL_PI;
    END_FBS
    EVENT_CONNECTIONS
      Gain100_0.CNF TO F_MUL_0_1.REQ;
      ReactorPressure_0.CNF TO r5_0.REQ;
      F_DIV_2_0.CNF TO yA_0.REQ;
      r4xFp_0.CNF TO CFeedRate_0.REQ;
      r2_1_0.CNF TO F_MUL_10_0.REQ;
      yAcontrolLoop14_0.INITO TO Delay_With_InitCondition_1.INIT;
      TIME2TIME_0_0.CNF TO E_CYCLE_1_0_0.START;
      NilaiK_0.CNF TO K_0_0.REQ;
      F_SUB_2.CNF TO r4_0.REQ;
      ProductionRate_0.INITO TO ReactorPressure_0.INIT;
      xmeas23x100_0.CNF TO F_DIV_2_0.REQ;
      xmeas7.CNF TO ReactorPressure_0.REQ;
      Server1.IND TO xmeas23.REQ;
      Server1.IND TO xmeas4.REQ;
      CFeedRate_0.CNF TO xmv4_0.REQ;
      yA_0.CNF TO yAcontrolLoop14_0.REQ;
      xmeas40.CNF TO GinProduct_0.REQ;
      Delay_With_InitCondition_0_0.CNF TO F_ADD_3_0.REQ;
      yAcontrolLoop14_0.INITO TO AFeedRate_0.INIT;
      r1_0.CNF TO r1xFp_0.REQ;
      xmeas3.CNF TO EFeedRate_0.REQ;
      r5_0.CNF TO F_MUL_0_0_0.REQ;
      SetpoxGain_0.CNF TO F_ADD_0_0_0.REQ;
      F_ADD_0_0_0.CNF TO Fp_0.REQ;
      Server1.IND TO xmeas25.REQ;
      ProdRatePIDoutputLREAL_0_0.CNF TO F_ADD_0_0_0.REQ;
      yAcontrolLoop14_0.CNF TO F_ADD_2_0.REQ;
      ProductionRate_0.CNF TO NilaiK_0.REQ;
      AFeedRate_0.CNF TO xmv3_0.REQ;
      xmeas23.CNF TO Gain100_0.REQ;
      yACcontrolLoop15_0.INITO TO yAcontrolLoop14_0.INIT;
      PurgeRate_0.CNF TO xmv6_0.REQ;
      xmv1_0.CNF TO E_CYCLE_1_0_0.START;
      DFeedRate_0.CNF TO xmv1_0.REQ;
      Server2.IND TO xmeas40.REQ;
      Fp_0.CNF TO r4xFp_0.REQ;
      Server2.IND TO xmeas17.REQ;
      AFeedRate_0.INITO TO CFeedRate_0.INIT;
      Server2.IND TO PctGsp_0.REQ;
      xmeas25.CNF TO F_ADD_0_1.REQ;
      F_MUL_10_0.CNF TO DFeedRate_0.REQ;
      K_0_0.CNF TO SetpoxGain_0.REQ;
      xmv6_0.CNF TO E_CYCLE_1_0_0.START;
      F_MUL_9_0.CNF TO EFeedRate_0.REQ;
      Fp_0.CNF TO F_MUL_10_0.REQ;
      ReactorPressure_0.INITO TO PurgeRate_0.INIT;
      DFeedRate_0.INITO TO yACcontrolLoop15_0.INIT;
      Fp_0.CNF TO r1xFp_0.REQ;
      Delay_With_InitCondition_1.CNF TO F_ADD_2_0.REQ;
      F_MUL_0_0_0.CNF TO PurgeRate_0.REQ;
      prodsetpointLREAL_0_0.CNF TO ProductionRate_0.REQ;
      F_ADD_2_0.CNF TO Delay_With_InitCondition_1.Start_and_REQ;
      ProductionRate_0.CNF TO ProdRatePIDoutputLREAL_0_0.REQ;
      xmv2_0.CNF TO E_CYCLE_1_0_0.START;
      F_MUL_0_1.CNF TO xmeas23x100_0.REQ;
      Fp_0.CNF TO F_MUL_0_0_0.REQ;
      xmv4_0.CNF TO E_CYCLE_1_0_0.START;
      E_CYCLE_1_0_0.EO TO Server2.RSP;
      yACcontrolLoop15_0.INITO TO Delay_With_InitCondition_0_0.INIT;
      Server2.IND TO xmeas7.REQ;
      F_ADD_3_0.CNF TO summmingpoinloop15_0.REQ;
      Server2.IND TO prodsetpointLREAL_0_0.REQ;
      yACcontrolLoop15_0.CNF TO F_ADD_3_0.REQ;
      F_ADD_0_1.CNF TO yAC_0.REQ;
      r3_1_0.CNF TO F_MUL_9_0.REQ;
      F_SUB_2.CNF TO Delay_With_InitCondition_0_0.Start_and_REQ;
      E_CYCLE_1_0_0.EO TO Server1.RSP;
      r4_0.CNF TO r4xFp_0.REQ;
      Server2.INITO TO ProductionRate_0.INIT;
      GinProduct_0.INITO TO EFeedRate_0.INIT;
      EFeedRate_0.CNF TO xmv2_0.REQ;
      yAC_0.CNF TO yACcontrolLoop15_0.REQ;
      xmeas17.CNF TO ProductionRate_0.REQ;
      Server2.IND TO xmeas3.REQ;
      Server2.IND TO xmeas10.REQ;
      r1xFp_0.CNF TO AFeedRate_0.REQ;
      Fp_0.CNF TO F_MUL_9_0.REQ;
      ProductionRate_0.CNF TO K_0_0.REQ;
      PurgeRate_0.INITO TO GinProduct_0.INIT;
      summmingpoinloop15_0.CNF TO F_SUB_2.REQ;
      F_ADD_2_0.CNF TO r1_0.REQ;
      xmeas4.CNF TO CFeedRate_0.REQ;
      xmv3_0.CNF TO E_CYCLE_1_0_0.START;
      Server1.INITO TO DFeedRate_0.INIT;
      xmeas10.CNF TO PurgeRate_0.REQ;
      PctGsp_0.CNF TO GinProduct_0.REQ;
      Feedforward.CNFr2 TO r2_1_0.REQ;
      Feedforward.CNFr3 TO r3_1_0.REQ;
      Fp_0.CNF TO Feedforward.RECFp;
      GinProduct_0.CNF TO Feedforward.RECEadj;
      PctGsp_0.CNF TO Feedforward.REQPctGsp;
      xmeas12.CNF TO SeparatorLevel.REQ;
      SeparatorLevel.CNF TO r6.REQ;
      Fp_0.CNF TO Fp.REQ;
      Fp.CNF TO F_MUL_1.REQ;
      r6.CNF TO F_MUL_1.REQ;
      xmeas14.CNF TO SeparatorFlowRate.REQ;
      F_MUL_1.CNF TO SeparatorFlowRate.REQ;
      SeparatorFlowRate.CNF TO xmv7.REQ;
      SeparatorLevel.INITO TO StripperLevel.INIT;
      StripperLevel.INITO TO SeparatorFlowRate.INIT;
      xmeas15.CNF TO StripperLevel.REQ;
      StripperLevel.CNF TO r7.REQ;
      r7.CNF TO F_MUL_1_0.REQ;
      Fp.CNF TO F_MUL_1_0.REQ;
      F_MUL_1_0.CNF TO StripperFlowRate.REQ;
      SeparatorFlowRate.INITO TO StripperFlowRate.INIT;
      StripperFlowRate.CNF TO xmv8.REQ;
      ReactorLevel.INITO TO SeparatorTemperature.INIT;
      SeparatorTemperature.INITO TO ReactorTemperature.INIT;
      xmeas8.CNF TO ReactorLevel.REQ;
      xmeas11.CNF TO SeparatorTemperature.REQ;
      ReactorLevel.CNF TO SeparatorTemperature.REQ;
      xmeas9.CNF TO ReactorTemperature.REQ;
      xmv7.CNF TO E_CYCLE_1_0_0.START;
      xmv8.CNF TO E_CYCLE_1_0_0.START;
      xmv11.CNF TO E_CYCLE_1_0_0.START;
      xmv10.CNF TO E_CYCLE_1_0_0.START;
      Server3.INITO TO SeparatorLevel.INIT;
      Server3.IND TO xmeas12.REQ;
      Server3.IND TO xmeas14.REQ;
      Server3.IND TO xmeas15.REQ;
      Server3.IND TO xmeas8.REQ;
      E_CYCLE_1_0_0.EO TO Server3.RSP;
      xmv5.CNF TO E_CYCLE_1_0_0.START;
      xmv9.CNF TO E_CYCLE_1_0_0.START;
      xmv12.CNF TO E_CYCLE_1_0_0.START;
      E_CYCLE_1_0_0.EO TO Server4.RSP;
      Server4.IND TO xmeas9.REQ;
      Server4.IND TO xmeas11.REQ;
      xmeas17.CNF TO xmeas17_2.REQ;
      Server3.IND TO xmeas17_2_0.REQ;
      xmeas17_2_0.CNF TO StripperFlowRate.REQ;
      ReactorTemperature.CNF TO xmv10.REQ;
      SeparatorTemperature.CNF TO xmv11.REQ;
      ReactorTemperature.CNF TO xmv5.REQ;
      ReactorTemperature.CNF TO xmv9.REQ;
      ReactorTemperature.CNF TO xmv12.REQ;
      EFeedRate_0.INITO TO ReactorLevel.INIT;
      Server1.IND TO DFeedRate_0.REQ;
      Server1.IND TO AFeedRate_0.REQ;
    END_CONNECTIONS
    DATA_CONNECTIONS
      xmeas17.OUT TO ProductionRate_0.ACTUAL;
      xmeas7.OUT TO ReactorPressure_0.ACTUAL;
      xmv3_0.OUT TO Server1.SD_2;
      Server2.RD_2 TO xmeas7.IN;
      Fp_0.OUT TO F_MUL_0_0_0.IN1;
      Fp_0.OUT TO r1xFp_0.IN2;
      Delay_With_InitCondition_0_0.LREAL1 TO F_ADD_3_0.IN2;
      Server2.RD_5 TO xmeas3.IN;
      r2_1_0.OUT TO F_MUL_10_0.IN1;
      xmeas23x100_0.OUT TO F_DIV_2_0.IN1;
      CFeedRate_0.OUT TO xmv4_0.IN;
      NilaiK_0.OUT TO K_0_0.IN2;
      Gain100_0.OUT TO F_MUL_0_1.IN2;
      DFeedRate_0.OUT TO xmv1_0.IN;
      F_MUL_0_0_0.OUT TO PurgeRate_0.SETPOINT;
      F_ADD_0_1.OUT TO yAC_0.IN;
      xmeas10.OUT TO PurgeRate_0.ACTUAL;
      PctGsp_0.OUT TO GinProduct_0.SETPOINT;
      r3_1_0.OUT TO F_MUL_9_0.IN1;
      Fp_0.OUT TO F_MUL_9_0.IN2;
      xmeas23.OUT TO F_ADD_0_1.IN1;
      xmeas40.OUT TO GinProduct_0.ACTUAL;
      ReactorPressure_0.OUT TO r5_0.IN;
      yACcontrolLoop15_0.DELTAOUTPUT TO F_ADD_3_0.IN1;
      F_ADD_2_0.OUT TO Delay_With_InitCondition_1.DelayedInput;
      TIME2TIME_0_0.OUT TO ProductionRate_0.SAMPLETIME;
      F_ADD_2_0.OUT TO r1_0.IN;
      ProductionRate_0.OUT TO ProdRatePIDoutputLREAL_0_0.IN;
      Delay_With_InitCondition_1.LREAL1 TO F_ADD_2_0.IN2;
      AFeedRate_0.OUT TO xmv3_0.IN;
      r1_0.OUT TO r1xFp_0.IN1;
      EFeedRate_0.OUT TO xmv2_0.IN;
      F_MUL_10_0.OUT TO DFeedRate_0.SETPOINT;
      F_MUL_9_0.OUT TO EFeedRate_0.SETPOINT;
      xmeas3.OUT TO EFeedRate_0.ACTUAL;
      xmeas23.OUT TO F_MUL_0_1.IN1;
      TIME2TIME_0_0.OUT TO E_CYCLE_1_0_0.DT;
      xmv4_0.OUT TO Server1.SD_3;
      TIME2TIME_0_0.OUT TO PurgeRate_0.SAMPLETIME;
      Server2.RD_3 TO xmeas10.IN;
      Server2.RD_4 TO xmeas40.IN;
      yAcontrolLoop14_0.DELTAOUTPUT TO F_SUB_2.IN2;
      F_SUB_2.OUT TO Delay_With_InitCondition_0_0.DelayedInput;
      F_SUB_2.OUT TO r4_0.IN;
      xmeas4.OUT TO CFeedRate_0.ACTUAL;
      xmeas25.OUT TO F_ADD_0_1.IN2;
      K_0_0.OUT TO SetpoxGain_0.IN;
      TIME2TIME_0_0.OUT TO DFeedRate_0.SAMPLETIME;
      F_MUL_0_1.OUT TO xmeas23x100_0.IN;
      xmv2_0.OUT TO Server2.SD_3;
      TIME2TIME_0_0.OUT TO ReactorPressure_0.SAMPLETIME;
      prodsetpointLREAL_0_0.OUT TO ProductionRate_0.SETPOINT;
      r1xFp_0.OUT TO AFeedRate_0.SETPOINT;
      yAC_0.OUT TO F_DIV_2_0.IN2;
      F_ADD_0_0_0.OUT TO Fp_0.IN;
      yAcontrolLoop14_0.DELTAOUTPUT TO F_ADD_2_0.IN1;
      ProdRatePIDoutputLREAL_0_0.OUT TO F_ADD_0_0_0.IN2;
      r4_0.OUT TO r4xFp_0.IN1;
      F_ADD_3_0.OUT TO summmingpoinloop15_0.IN;
      SetpoxGain_0.OUT TO F_ADD_0_0_0.IN1;
      TIME2TIME_0_0.OUT TO GinProduct_0.SAMPLETIME;
      Server1.RD_5 TO xmeas4.IN;
      r4xFp_0.OUT TO CFeedRate_0.SETPOINT;
      Server1.RD_3 TO xmeas25.IN;
      yAC_0.OUT TO yACcontrolLoop15_0.ACTUAL;
      PurgeRate_0.OUT TO xmv6_0.IN;
      r5_0.OUT TO F_MUL_0_0_0.IN2;
      xmv6_0.OUT TO Server2.SD_1;
      xmv6_0.OUT TO Server2.SD_2;
      Server2.RD_1 TO xmeas17.IN;
      yA_0.OUT TO yAcontrolLoop14_0.ACTUAL;
      Server1.RD_2 TO xmeas23.IN;
      xmv1_0.OUT TO Server1.SD_1;
      F_DIV_2_0.OUT TO yA_0.IN;
      ProdRatePIDoutputLREAL_0_0.OUT TO K_0_0.IN1;
      summmingpoinloop15_0.OUT TO F_SUB_2.IN1;
      TIME2TIME_0_0.OUT TO EFeedRate_0.SAMPLETIME;
      Fp_0.OUT TO r4xFp_0.IN2;
      Fp_0.OUT TO F_MUL_10_0.IN2;
      Feedforward.r2 TO r2_1_0.IN;
      Feedforward.r3 TO r3_1_0.IN;
      Fp_0.OUT TO Feedforward.Fp;
      GinProduct_0.OUT TO Feedforward.Eadj;
      PctGsp_0.OUT TO Feedforward.PctGsp;
      xmeas12.OUT TO SeparatorLevel.ACTUAL;
      TIME2TIME_0_0.OUT TO SeparatorLevel.SAMPLETIME;
      SeparatorLevel.OUT TO r6.IN;
      Fp_0.OUT TO Fp.IN;
      Fp.OUT TO F_MUL_1.IN1;
      r6.OUT TO F_MUL_1.IN2;
      xmeas14.OUT TO SeparatorFlowRate.ACTUAL;
      F_MUL_1.OUT TO SeparatorFlowRate.SETPOINT;
      SeparatorFlowRate.OUT TO xmv7.IN;
      xmeas15.OUT TO StripperLevel.ACTUAL;
      TIME2TIME_0_0.OUT TO SeparatorFlowRate.SAMPLETIME;
      TIME2TIME_0_0.OUT TO StripperLevel.SAMPLETIME;
      StripperLevel.OUT TO r7.IN;
      r7.OUT TO F_MUL_1_0.IN1;
      Fp.OUT TO F_MUL_1_0.IN2;
      F_MUL_1_0.OUT TO StripperFlowRate.SETPOINT;
      TIME2TIME_0_0.OUT TO StripperFlowRate.SAMPLETIME;
      StripperFlowRate.OUT TO xmv8.IN;
      xmeas8.OUT TO ReactorLevel.ACTUAL;
      ReactorLevel.OUT TO SeparatorTemperature.SETPOINT;
      xmeas11.OUT TO SeparatorTemperature.ACTUAL;
      SeparatorTemperature.OUT TO xmv11.IN;
      xmeas9.OUT TO ReactorTemperature.ACTUAL;
      ReactorTemperature.OUT TO xmv10.IN;
      xmv7.OUT TO Server3.SD_1;
      Server3.RD_1 TO xmeas12.IN;
      Server3.RD_2 TO xmeas14.IN;
      Server3.RD_3 TO xmeas15.IN;
      Server3.RD_5 TO xmeas8.IN;
      xmv8.OUT TO Server3.SD_2;
      xmv11.OUT TO Server3.SD_3;
      xmv10.OUT TO Server4.SD_1;
      TIME2TIME_0_0.OUT TO ReactorLevel.SAMPLETIME;
      TIME2TIME_0_0.OUT TO ReactorTemperature.SAMPLETIME;
      TIME2TIME_0_0.OUT TO SeparatorTemperature.SAMPLETIME;
      xmv5.OUT TO Server4.SD_2;
      xmv9.OUT TO Server4.SD_3;
      xmv12.OUT TO Server4.SD_4;
      Server4.RD_1 TO xmeas11.IN;
      Server4.RD_2 TO xmeas9.IN;
      xmeas17.OUT TO xmeas17_2.IN;
      TIME2TIME_0_0.OUT TO AFeedRate_0.SAMPLETIME;
      TIME2TIME_0_0.OUT TO CFeedRate_0.SAMPLETIME;
      xmeas17_2_0.OUT TO StripperFlowRate.ACTUAL;
      Server1.RD_1 TO DFeedRate_0.ACTUAL;
      Server1.RD_4 TO AFeedRate_0.ACTUAL;
    END_CONNECTIONS
  END_APPLICATION
  APPLICATION pressureloop
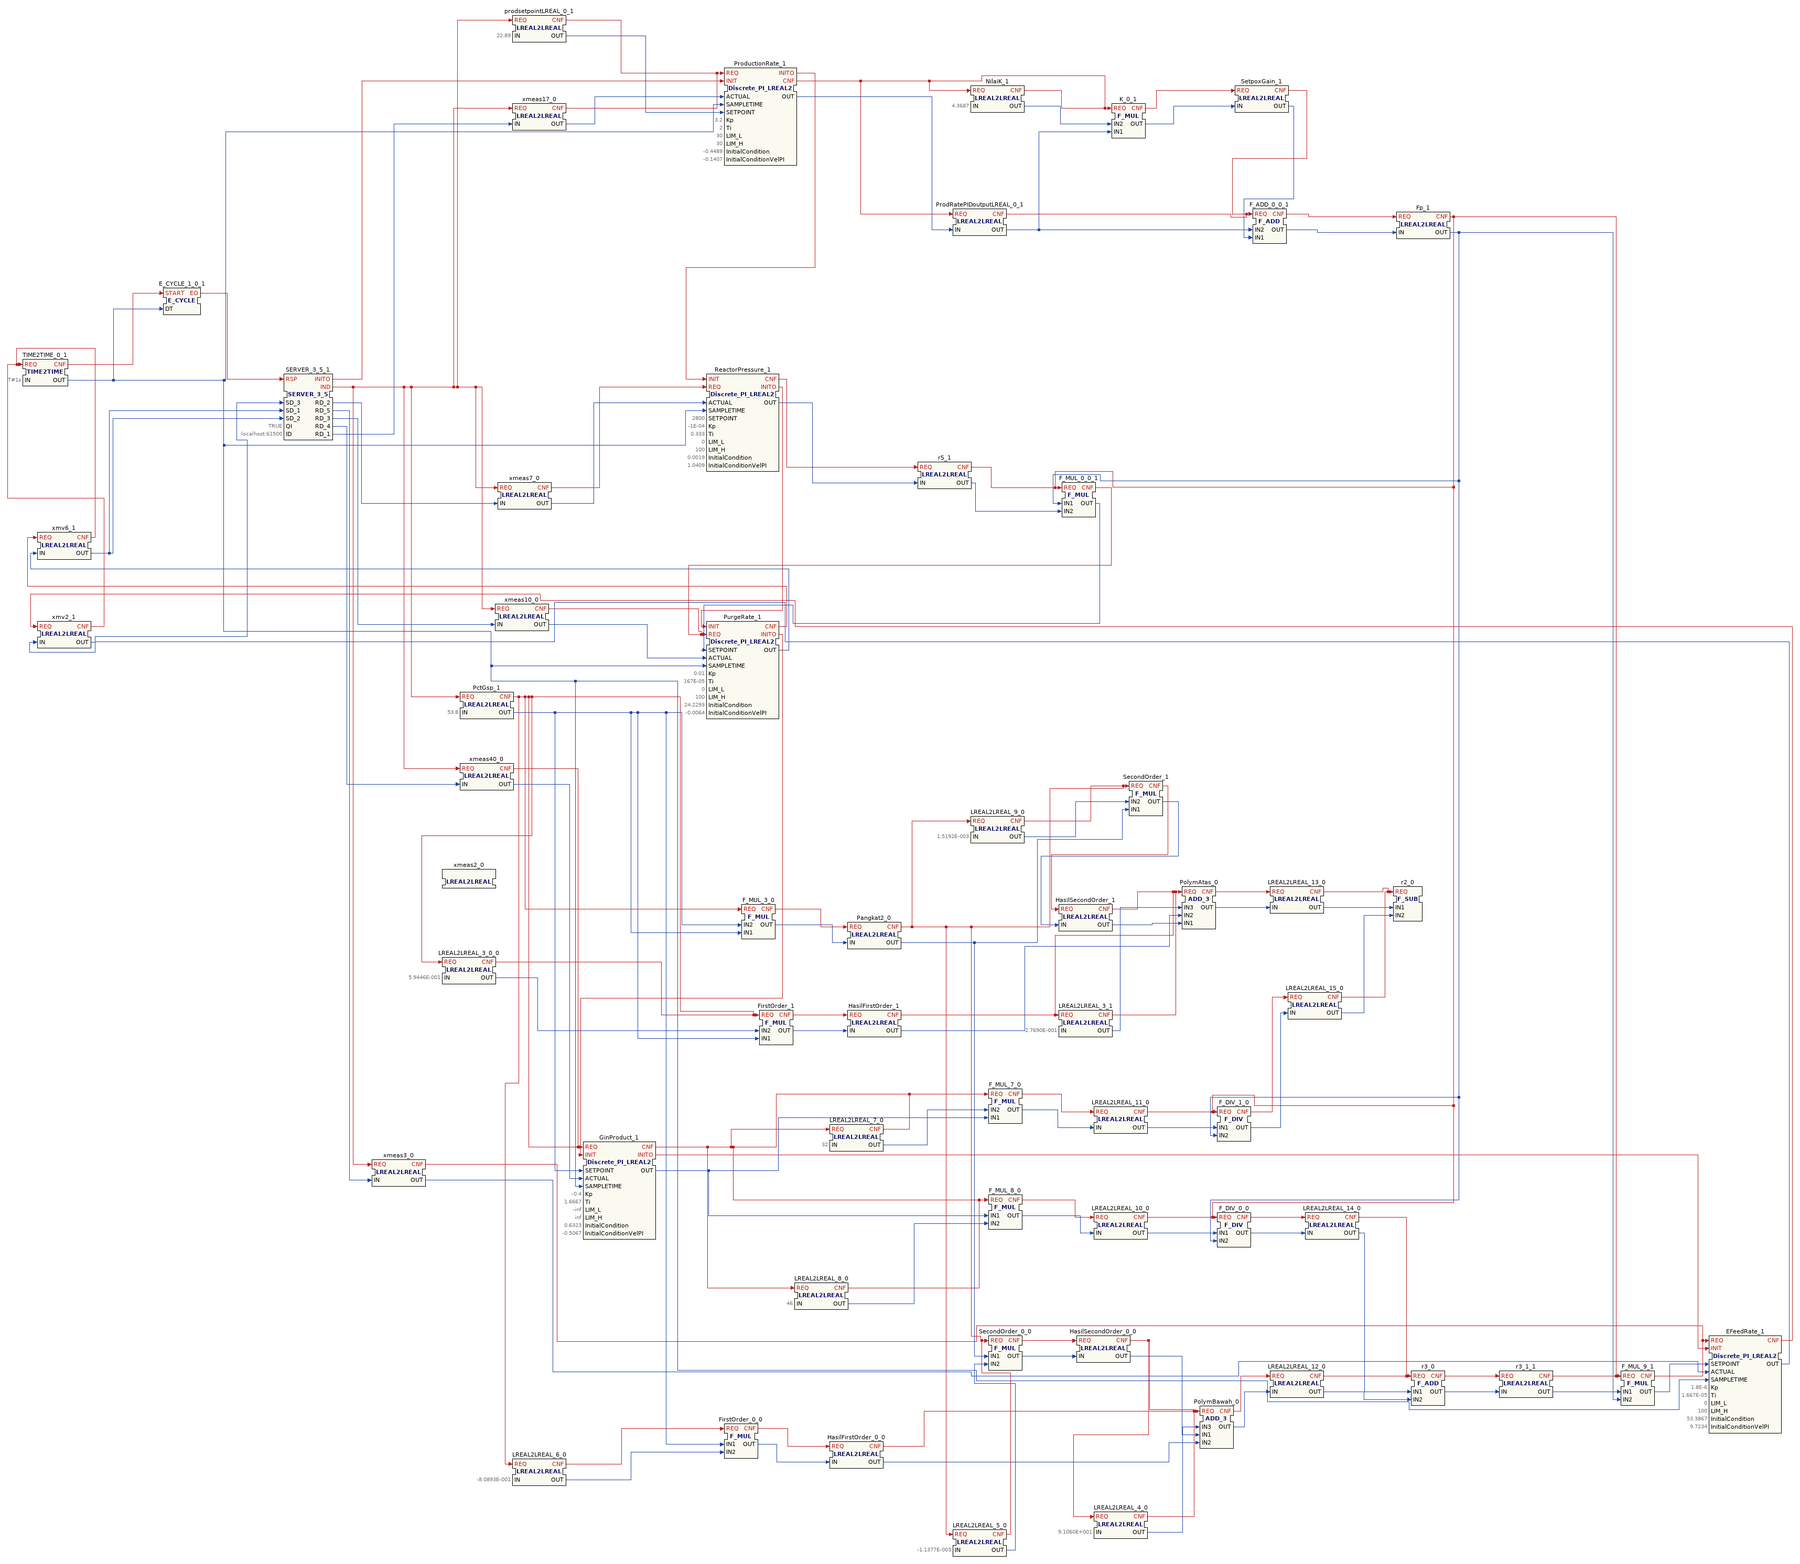
    FBS
      xmeas17_0 : LREAL2LREAL;
      ProdRatePIDoutputLREAL_0_1 : LREAL2LREAL;
      K_0_1 : F_MUL;
      prodsetpointLREAL_0_1 : LREAL2LREAL(IN := 22.89);
      F_ADD_0_0_1 : F_ADD;
      F_MUL_0_0_1 : F_MUL;
      E_CYCLE_1_0_1 : E_CYCLE;
      xmeas7_0 : LREAL2LREAL;
      xmeas10_0 : LREAL2LREAL;
      SetpoxGain_1 : LREAL2LREAL;
      Fp_1 : LREAL2LREAL;
      r5_1 : LREAL2LREAL;
      NilaiK_1 : LREAL2LREAL(IN := 4.3687);
      SERVER_3_5_1 : SERVER_3_5(QI := TRUE, ID := localhost:61500);
      PctGsp_1 : LREAL2LREAL(IN := 53.8);
      xmv6_1 : LREAL2LREAL;
      PolymAtas_0 : ADD_3;
      F_MUL_3_0 : F_MUL;
      FirstOrder_1 : F_MUL;
      SecondOrder_1 : F_MUL;
      Pangkat2_0 : LREAL2LREAL;
      HasilSecondOrder_1 : LREAL2LREAL;
      HasilFirstOrder_1 : LREAL2LREAL;
      SecondOrder_0_0 : F_MUL;
      HasilSecondOrder_0_0 : LREAL2LREAL;
      FirstOrder_0_0 : F_MUL;
      HasilFirstOrder_0_0 : LREAL2LREAL;
      PolymBawah_0 : ADD_3;
      F_MUL_7_0 : F_MUL;
      F_MUL_8_0 : F_MUL;
      LREAL2LREAL_10_0 : LREAL2LREAL;
      LREAL2LREAL_11_0 : LREAL2LREAL;
      F_DIV_0_0 : F_DIV;
      LREAL2LREAL_12_0 : LREAL2LREAL;
      LREAL2LREAL_13_0 : LREAL2LREAL;
      r3_0 : F_ADD;
      r2_0 : F_SUB;
      LREAL2LREAL_14_0 : LREAL2LREAL;
      F_DIV_1_0 : F_DIV;
      LREAL2LREAL_15_0 : LREAL2LREAL;
      r3_1_1 : LREAL2LREAL;
      F_MUL_9_1 : F_MUL;
      xmeas40_0 : LREAL2LREAL;
      xmeas3_0 : LREAL2LREAL;
      xmv2_1 : LREAL2LREAL;
      ProductionRate_1 : Discrete_PI_LREAL2(Kp := 3.2, Ti := 2, LIM_L := 30, LIM_H := 30, InitialCondition := -0.4489, InitialConditionVelPI := -0.1407);
      ReactorPressure_1 : Discrete_PI_LREAL2(SETPOINT := 2800, Kp := -1E-04, Ti := 0.333, LIM_L := 0, LIM_H := 100, InitialCondition := 0.0019, InitialConditionVelPI := 1.0409);
      PurgeRate_1 : Discrete_PI_LREAL2(Kp := 0.01, Ti := 167E-05, LIM_L := 0, LIM_H := 100, InitialCondition := 24.2293, InitialConditionVelPI := -0.0064);
      GinProduct_1 : Discrete_PI_LREAL2(Kp := -0.4, Ti := 1.6667, LIM_L := -inf, LIM_H := inf, InitialCondition := 0.6323, InitialConditionVelPI := -0.5067);
      EFeedRate_1 : Discrete_PI_LREAL2(Kp := 1.8E-6, Ti := 1.667E-05, LIM_L := 0, LIM_H := 100, InitialCondition := 53.3867, InitialConditionVelPI := 9.7234);
      TIME2TIME_0_1 : TIME2TIME(IN := T#1s);
      LREAL2LREAL_3_1 : LREAL2LREAL(IN := 2.7690E-001);
      LREAL2LREAL_3_0_0 : LREAL2LREAL(IN := 5.9446E-001);
      LREAL2LREAL_5_0 : LREAL2LREAL(IN := -1.1377E-003);
      LREAL2LREAL_6_0 : LREAL2LREAL(IN := -8.0893E-001);
      LREAL2LREAL_4_0 : LREAL2LREAL(IN := 9.1060E+001);
      LREAL2LREAL_7_0 : LREAL2LREAL(IN := 32);
      LREAL2LREAL_8_0 : LREAL2LREAL(IN := 46);
      LREAL2LREAL_9_0 : LREAL2LREAL(IN := 1.5192E-003);
      xmeas2_0 : LREAL2LREAL;
    END_FBS
    EVENT_CONNECTIONS
      ReactorPressure_1.CNF TO r5_1.REQ;
      PctGsp_1.CNF TO F_MUL_3_0.REQ;
      PctGsp_1.CNF TO GinProduct_1.REQ;
      PolymAtas_0.CNF TO LREAL2LREAL_13_0.REQ;
      HasilSecondOrder_0_0.CNF TO LREAL2LREAL_4_0.REQ;
      LREAL2LREAL_7_0.CNF TO F_MUL_7_0.REQ;
      FirstOrder_0_0.CNF TO HasilFirstOrder_0_0.REQ;
      PolymBawah_0.CNF TO LREAL2LREAL_12_0.REQ;
      NilaiK_1.CNF TO K_0_1.REQ;
      HasilFirstOrder_0_0.CNF TO PolymBawah_0.REQ;
      ProductionRate_1.INITO TO ReactorPressure_1.INIT;
      xmeas7_0.CNF TO ReactorPressure_1.REQ;
      GinProduct_1.CNF TO LREAL2LREAL_8_0.REQ;
      LREAL2LREAL_6_0.CNF TO FirstOrder_0_0.REQ;
      r3_0.CNF TO r3_1_1.REQ;
      xmeas40_0.CNF TO GinProduct_1.REQ;
      LREAL2LREAL_9_0.CNF TO SecondOrder_1.REQ;
      Pangkat2_0.CNF TO LREAL2LREAL_9_0.REQ;
      F_DIV_1_0.CNF TO LREAL2LREAL_15_0.REQ;
      GinProduct_1.CNF TO F_MUL_8_0.REQ;
      FirstOrder_1.CNF TO HasilFirstOrder_1.REQ;
      LREAL2LREAL_15_0.CNF TO r2_0.REQ;
      PctGsp_1.CNF TO LREAL2LREAL_3_0_0.REQ;
      xmeas3_0.CNF TO EFeedRate_1.REQ;
      LREAL2LREAL_12_0.CNF TO r3_0.REQ;
      r5_1.CNF TO F_MUL_0_0_1.REQ;
      Pangkat2_0.CNF TO SecondOrder_0_0.REQ;
      F_MUL_3_0.CNF TO Pangkat2_0.REQ;
      SetpoxGain_1.CNF TO F_ADD_0_0_1.REQ;
      F_MUL_8_0.CNF TO LREAL2LREAL_10_0.REQ;
      HasilFirstOrder_1.CNF TO LREAL2LREAL_3_1.REQ;
      F_ADD_0_0_1.CNF TO Fp_1.REQ;
      ProdRatePIDoutputLREAL_0_1.CNF TO F_ADD_0_0_1.REQ;
      Pangkat2_0.CNF TO LREAL2LREAL_5_0.REQ;
      ProductionRate_1.CNF TO NilaiK_1.REQ;
      F_DIV_0_0.CNF TO LREAL2LREAL_14_0.REQ;
      PurgeRate_1.CNF TO xmv6_1.REQ;
      HasilSecondOrder_1.CNF TO PolymAtas_0.REQ;
      LREAL2LREAL_8_0.CNF TO F_MUL_8_0.REQ;
      Fp_1.CNF TO F_DIV_0_0.REQ;
      LREAL2LREAL_14_0.CNF TO r3_0.REQ;
      SecondOrder_1.CNF TO HasilSecondOrder_1.REQ;
      F_MUL_7_0.CNF TO LREAL2LREAL_11_0.REQ;
      LREAL2LREAL_3_0_0.CNF TO FirstOrder_1.REQ;
      K_0_1.CNF TO SetpoxGain_1.REQ;
      PctGsp_1.CNF TO FirstOrder_1.REQ;
      F_MUL_9_1.CNF TO EFeedRate_1.REQ;
      PctGsp_1.CNF TO LREAL2LREAL_6_0.REQ;
      ReactorPressure_1.INITO TO PurgeRate_1.INIT;
      Fp_1.CNF TO F_DIV_1_0.REQ;
      SecondOrder_0_0.CNF TO HasilSecondOrder_0_0.REQ;
      F_MUL_0_0_1.CNF TO PurgeRate_1.REQ;
      LREAL2LREAL_13_0.CNF TO r2_0.REQ;
      prodsetpointLREAL_0_1.CNF TO ProductionRate_1.REQ;
      LREAL2LREAL_4_0.CNF TO PolymBawah_0.REQ;
      ProductionRate_1.CNF TO ProdRatePIDoutputLREAL_0_1.REQ;
      Fp_1.CNF TO F_MUL_0_0_1.REQ;
      Pangkat2_0.CNF TO SecondOrder_1.REQ;
      LREAL2LREAL_11_0.CNF TO F_DIV_1_0.REQ;
      r3_1_1.CNF TO F_MUL_9_1.REQ;
      LREAL2LREAL_3_1.CNF TO PolymAtas_0.REQ;
      GinProduct_1.INITO TO EFeedRate_1.INIT;
      LREAL2LREAL_5_0.CNF TO SecondOrder_0_0.REQ;
      GinProduct_1.CNF TO LREAL2LREAL_7_0.REQ;
      EFeedRate_1.CNF TO xmv2_1.REQ;
      GinProduct_1.CNF TO F_MUL_7_0.REQ;
      xmeas17_0.CNF TO ProductionRate_1.REQ;
      Fp_1.CNF TO F_MUL_9_1.REQ;
      ProductionRate_1.CNF TO K_0_1.REQ;
      HasilSecondOrder_0_0.CNF TO PolymBawah_0.REQ;
      PurgeRate_1.INITO TO GinProduct_1.INIT;
      HasilFirstOrder_1.CNF TO PolymAtas_0.REQ;
      LREAL2LREAL_10_0.CNF TO F_DIV_0_0.REQ;
      xmeas10_0.CNF TO PurgeRate_1.REQ;
      xmv2_1.CNF TO TIME2TIME_0_1.REQ;
      xmv6_1.CNF TO TIME2TIME_0_1.REQ;
      SERVER_3_5_1.INITO TO ProductionRate_1.INIT;
      SERVER_3_5_1.IND TO xmeas17_0.REQ;
      SERVER_3_5_1.IND TO prodsetpointLREAL_0_1.REQ;
      SERVER_3_5_1.IND TO xmeas7_0.REQ;
      SERVER_3_5_1.IND TO xmeas10_0.REQ;
      SERVER_3_5_1.IND TO xmeas40_0.REQ;
      SERVER_3_5_1.IND TO xmeas3_0.REQ;
      SERVER_3_5_1.IND TO PctGsp_1.REQ;
      E_CYCLE_1_0_1.EO TO SERVER_3_5_1.RSP;
      TIME2TIME_0_1.CNF TO E_CYCLE_1_0_1.START;
    END_CONNECTIONS
    DATA_CONNECTIONS
      xmeas17_0.OUT TO ProductionRate_1.ACTUAL;
      LREAL2LREAL_7_0.OUT TO F_MUL_7_0.IN2;
      xmeas7_0.OUT TO ReactorPressure_1.ACTUAL;
      LREAL2LREAL_9_0.OUT TO SecondOrder_1.IN2;
      SERVER_3_5_1.RD_2 TO xmeas7_0.IN;
      Fp_1.OUT TO F_MUL_0_0_1.IN1;
      SERVER_3_5_1.RD_5 TO xmeas3_0.IN;
      SecondOrder_1.OUT TO HasilSecondOrder_1.IN;
      PctGsp_1.OUT TO FirstOrder_0_0.IN1;
      SecondOrder_0_0.OUT TO HasilSecondOrder_0_0.IN;
      F_DIV_0_0.OUT TO LREAL2LREAL_14_0.IN;
      F_MUL_3_0.OUT TO Pangkat2_0.IN;
      NilaiK_1.OUT TO K_0_1.IN2;
      PolymAtas_0.OUT TO LREAL2LREAL_13_0.IN;
      GinProduct_1.OUT TO F_MUL_8_0.IN1;
      LREAL2LREAL_14_0.OUT TO r3_0.IN1;
      F_MUL_0_0_1.OUT TO PurgeRate_1.SETPOINT;
      PctGsp_1.OUT TO F_MUL_3_0.IN2;
      PctGsp_1.OUT TO F_MUL_3_0.IN1;
      xmeas10_0.OUT TO PurgeRate_1.ACTUAL;
      PctGsp_1.OUT TO GinProduct_1.SETPOINT;
      r3_1_1.OUT TO F_MUL_9_1.IN1;
      Fp_1.OUT TO F_MUL_9_1.IN2;
      LREAL2LREAL_4_0.OUT TO PolymBawah_0.IN3;
      xmeas40_0.OUT TO GinProduct_1.ACTUAL;
      LREAL2LREAL_11_0.OUT TO F_DIV_1_0.IN1;
      ReactorPressure_1.OUT TO r5_1.IN;
      LREAL2LREAL_3_1.OUT TO PolymAtas_0.IN3;
      F_MUL_8_0.OUT TO LREAL2LREAL_10_0.IN;
      TIME2TIME_0_1.OUT TO ProductionRate_1.SAMPLETIME;
      LREAL2LREAL_10_0.OUT TO F_DIV_0_0.IN1;
      ProductionRate_1.OUT TO ProdRatePIDoutputLREAL_0_1.IN;
      r3_0.OUT TO r3_1_1.IN;
      GinProduct_1.OUT TO F_MUL_7_0.IN1;
      FirstOrder_0_0.OUT TO HasilFirstOrder_0_0.IN;
      EFeedRate_1.OUT TO xmv2_1.IN;
      F_MUL_9_1.OUT TO EFeedRate_1.SETPOINT;
      xmeas3_0.OUT TO EFeedRate_1.ACTUAL;
      LREAL2LREAL_13_0.OUT TO r2_0.IN1;
      HasilSecondOrder_0_0.OUT TO PolymBawah_0.IN1;
      TIME2TIME_0_1.OUT TO E_CYCLE_1_0_1.DT;
      TIME2TIME_0_1.OUT TO PurgeRate_1.SAMPLETIME;
      Pangkat2_0.OUT TO SecondOrder_0_0.IN1;
      SERVER_3_5_1.RD_3 TO xmeas10_0.IN;
      Fp_1.OUT TO F_DIV_1_0.IN2;
      SERVER_3_5_1.RD_4 TO xmeas40_0.IN;
      FirstOrder_1.OUT TO HasilFirstOrder_1.IN;
      HasilFirstOrder_1.OUT TO PolymAtas_0.IN2;
      LREAL2LREAL_12_0.OUT TO r3_0.IN2;
      K_0_1.OUT TO SetpoxGain_1.IN;
      LREAL2LREAL_6_0.OUT TO FirstOrder_0_0.IN2;
      LREAL2LREAL_5_0.OUT TO SecondOrder_0_0.IN2;
      xmv2_1.OUT TO SERVER_3_5_1.SD_3;
      TIME2TIME_0_1.OUT TO ReactorPressure_1.SAMPLETIME;
      prodsetpointLREAL_0_1.OUT TO ProductionRate_1.SETPOINT;
      Pangkat2_0.OUT TO SecondOrder_1.IN1;
      F_ADD_0_0_1.OUT TO Fp_1.IN;
      ProdRatePIDoutputLREAL_0_1.OUT TO F_ADD_0_0_1.IN2;
      TIME2TIME_0_1.OUT TO EFeedRate_1.SAMPLETIME;
      SetpoxGain_1.OUT TO F_ADD_0_0_1.IN1;
      TIME2TIME_0_1.OUT TO GinProduct_1.SAMPLETIME;
      LREAL2LREAL_3_0_0.OUT TO FirstOrder_1.IN2;
      Fp_1.OUT TO F_DIV_0_0.IN2;
      F_MUL_7_0.OUT TO LREAL2LREAL_11_0.IN;
      PurgeRate_1.OUT TO xmv6_1.IN;
      r5_1.OUT TO F_MUL_0_0_1.IN2;
      xmv6_1.OUT TO SERVER_3_5_1.SD_1;
      xmv6_1.OUT TO SERVER_3_5_1.SD_2;
      HasilSecondOrder_1.OUT TO PolymAtas_0.IN1;
      SERVER_3_5_1.RD_1 TO xmeas17_0.IN;
      F_DIV_1_0.OUT TO LREAL2LREAL_15_0.IN;
      LREAL2LREAL_8_0.OUT TO F_MUL_8_0.IN2;
      PolymBawah_0.OUT TO LREAL2LREAL_12_0.IN;
      HasilFirstOrder_0_0.OUT TO PolymBawah_0.IN2;
      PctGsp_1.OUT TO FirstOrder_1.IN1;
      ProdRatePIDoutputLREAL_0_1.OUT TO K_0_1.IN1;
      LREAL2LREAL_15_0.OUT TO r2_0.IN2;
    END_CONNECTIONS
  END_APPLICATION
  APPLICATION reactortemperatureloop
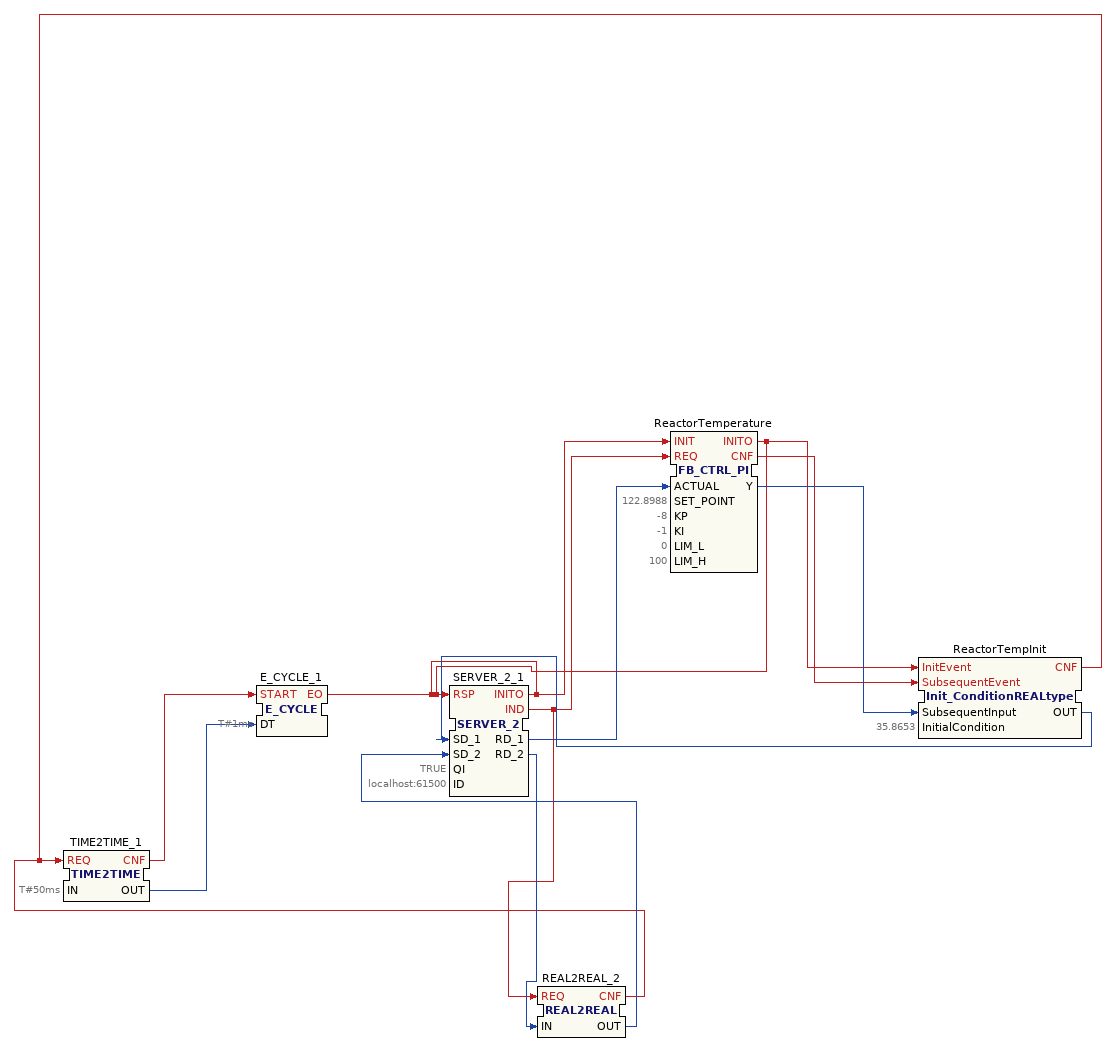
    FBS
      TIME2TIME_1 : TIME2TIME(IN := T#50ms);
      E_CYCLE_1 : E_CYCLE(DT := T#1ms);
      SERVER_2_1 : SERVER_2(QI := TRUE, ID := localhost:61500);
      ReactorTemperature : FB_CTRL_PI(SET_POINT := 122.8988, KP := -8, KI := -1, LIM_L := 0, LIM_H := 100);
      ReactorTempInit : Init_ConditionREALtype(InitialCondition := 35.8653);
      REAL2REAL_2 : REAL2REAL;
    END_FBS
    EVENT_CONNECTIONS
      TIME2TIME_1.CNF TO E_CYCLE_1.START;
      E_CYCLE_1.EO TO SERVER_2_1.RSP;
      ReactorTemperature.INITO TO SERVER_2_1.RSP;
      SERVER_2_1.INITO TO ReactorTemperature.INIT;
      SERVER_2_1.IND TO ReactorTemperature.REQ;
      ReactorTemperature.INITO TO ReactorTempInit.InitEvent;
      ReactorTemperature.CNF TO ReactorTempInit.SubsequentEvent;
      ReactorTempInit.CNF TO TIME2TIME_1.REQ;
      SERVER_2_1.IND TO REAL2REAL_2.REQ;
      REAL2REAL_2.CNF TO TIME2TIME_1.REQ;
      SERVER_2_1.INITO TO SERVER_2_1.RSP;
    END_CONNECTIONS
    DATA_CONNECTIONS
      TIME2TIME_1.OUT TO E_CYCLE_1.DT;
      SERVER_2_1.RD_1 TO ReactorTemperature.ACTUAL;
      ReactorTemperature.Y TO ReactorTempInit.SubsequentInput;
      ReactorTempInit.OUT TO SERVER_2_1.SD_1;
      SERVER_2_1.RD_2 TO REAL2REAL_2.IN;
      REAL2REAL_2.OUT TO SERVER_2_1.SD_2;
    END_CONNECTIONS
  END_APPLICATION
  APPLICATION reactortemperatureloopconvertin4diac
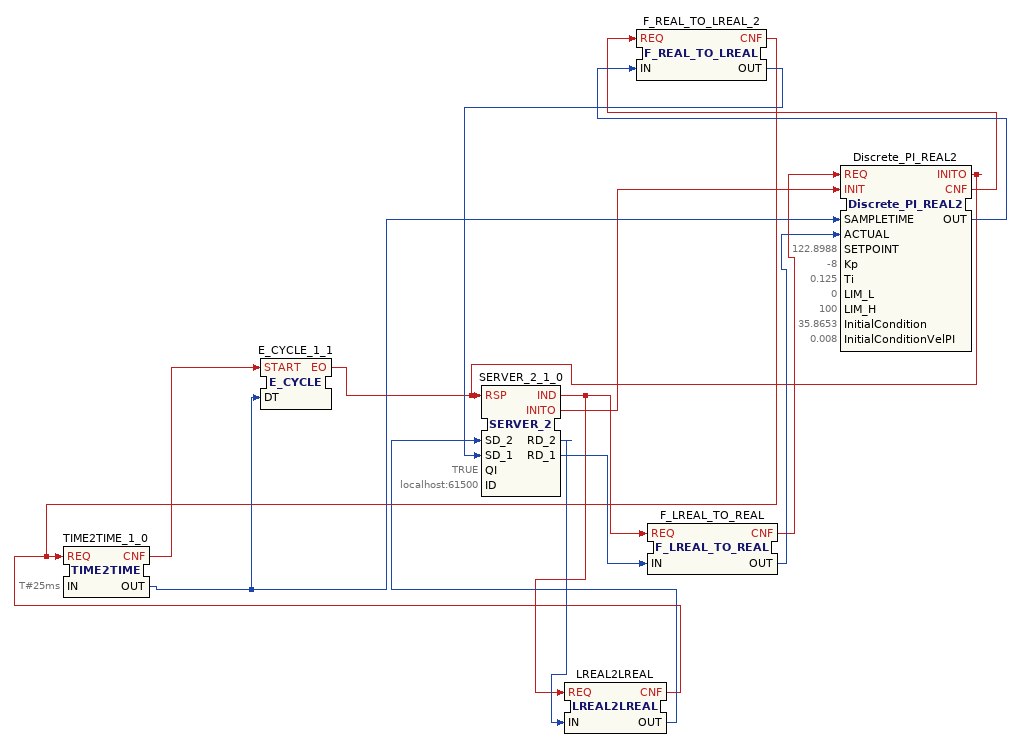
    FBS
      TIME2TIME_1_0 : TIME2TIME(IN := T#25ms);
      E_CYCLE_1_1 : E_CYCLE;
      SERVER_2_1_0 : SERVER_2(QI := TRUE, ID := localhost:61500);
      LREAL2LREAL : LREAL2LREAL;
      Discrete_PI_REAL2 : Discrete_PI_REAL2(SETPOINT := 122.8988, Kp := -8, Ti := 0.125, LIM_L := 0, LIM_H := 100, InitialCondition := 35.8653, InitialConditionVelPI := 0.008);
      F_LREAL_TO_REAL : F_LREAL_TO_REAL;
      F_REAL_TO_LREAL_2 : F_REAL_TO_LREAL;
    END_FBS
    EVENT_CONNECTIONS
      E_CYCLE_1_1.EO TO SERVER_2_1_0.RSP;
      TIME2TIME_1_0.CNF TO E_CYCLE_1_1.START;
      SERVER_2_1_0.IND TO LREAL2LREAL.REQ;
      LREAL2LREAL.CNF TO TIME2TIME_1_0.REQ;
      F_LREAL_TO_REAL.CNF TO Discrete_PI_REAL2.REQ;
      SERVER_2_1_0.IND TO F_LREAL_TO_REAL.REQ;
      SERVER_2_1_0.INITO TO Discrete_PI_REAL2.INIT;
      Discrete_PI_REAL2.INITO TO SERVER_2_1_0.RSP;
      Discrete_PI_REAL2.CNF TO F_REAL_TO_LREAL_2.REQ;
      F_REAL_TO_LREAL_2.CNF TO TIME2TIME_1_0.REQ;
    END_CONNECTIONS
    DATA_CONNECTIONS
      TIME2TIME_1_0.OUT TO E_CYCLE_1_1.DT;
      SERVER_2_1_0.RD_2 TO LREAL2LREAL.IN;
      LREAL2LREAL.OUT TO SERVER_2_1_0.SD_2;
      TIME2TIME_1_0.OUT TO Discrete_PI_REAL2.SAMPLETIME;
      SERVER_2_1_0.RD_1 TO F_LREAL_TO_REAL.IN;
      F_LREAL_TO_REAL.OUT TO Discrete_PI_REAL2.ACTUAL;
      Discrete_PI_REAL2.OUT TO F_REAL_TO_LREAL_2.IN;
      F_REAL_TO_LREAL_2.OUT TO SERVER_2_1_0.SD_1;
    END_CONNECTIONS
  END_APPLICATION
  APPLICATION plantwide
    FBS
      ProductionRate : FB_CTRL_PI(KP := 3.2, KI := 6.4, LIM_L := -30, LIM_H := 30);
      ProductionSetpoint : REAL2REAL(IN := 22.89);
      F_MUL_2 : F_MUL(IN2 := 4.36871996);
      Fp_ : F_ADD;
      KxProdSetpoint : REAL2REAL;
      yAcontrol : FB_CTRL_PI(SET_POINT := 63.13725, KP := 2.00E-04, KI := 0.0002);
      yACcontrol : FB_CTRL_PI(SET_POINT := 51, KP := 3.00E-04, KI := 0.0002);
      AandCControl : SERVER_0_2(QI := TRUE, ID := localhost:61000);
      E_CYCLE_3 : E_CYCLE(DT := T#0.1s);
      xmeas23 : REAL2REAL;
      F_MUL_4 : F_MUL(IN2 := 100);
      yAC : F_ADD;
      yA : F_DIV;
      xmeas25 : REAL2REAL;
      xmeas23_2 : REAL2REAL;
      yAC_ : REAL2REAL;
      yA_ : REAL2REAL;
      F_SUB_0 : F_SUB;
      Loop15 : REAL2REAL;
      F_ADD_4 : F_ADD;
      Delay_With_InitConditionREALtype : Delay_With_InitConditionREALtype(DelayTime := T#0.1s, InitialCondition := 0.092236609900323);
      r4 : REAL2REAL;
      F_ADD_5 : F_ADD;
      r1 : REAL2REAL;
      Delay_With_InitConditionREALtype_0 : Delay_With_InitConditionREALtype(DelayTime := T#0.1s, InitialCondition := 0.002722836244293);
      TIME2TIME_2 : TIME2TIME(IN := T#100ms);
      CFeedRate : FB_CTRL_PI(KP := 0.003, KI := 0, LIM_L := 0, LIM_H := 100);
      AFeedRate : FB_CTRL_PI(KP := 0.01, KI := 0, LIM_L := 0, LIM_H := 100);
      Fp : REAL2REAL;
      AFeedRateSetpoint : F_MUL;
      CFeedRateSetpoint : F_MUL;
      GinProduct : FB_CTRL_PI(KP := -0.4, KI := -0.666666667, LIM_L := -100000000000, LIM_H := 100000000000);
      MoleGSetpoint : REAL2REAL(IN := 53.8);
      FeedforwardREAL : FeedforwardREAL;
      DFeedRateSetpoint : F_MUL;
      DFeedRate : FB_CTRL_PI(KP := 1.60E-06, KI := 0, LIM_L := 0, LIM_H := 100);
      EFeedRateSetpoint : F_MUL;
      EFeedRate : FB_CTRL_PI(KP := 1.80E-06, KI := 0, LIM_L := 0, LIM_H := 100);
      r5 : F_MUL;
      r7 : F_MUL;
      r6 : F_MUL;
      SeparatorLeel : FB_CTRL_PI(SET_POINT := 50, KP := -1.00E-03, KI := 0, LIM_L := 0, LIM_H := 100);
      RectorPressure : FB_CTRL_PI(SET_POINT := 2800, KP := -1.00E-04, KI := 0, LIM_L := 0, LIM_H := 100);
      StripperLevel : FB_CTRL_PI(SET_POINT := 50, KP := -2.00E-04, KI := -0.000666667, LIM_L := 0, LIM_H := 100);
      PurgeRate : FB_CTRL_PI(KP := 0.01, KI := 0, LIM_L := 0, LIM_H := 100);
      SeparatorFlowRate : FB_CTRL_PI(KP := 4.00E-04, KI := 0, LIM_L := 0, LIM_H := 100);
      StripperFlowRate : FB_CTRL_PI(KP := 4.00E-04, KI := 0, LIM_L := 0, LIM_H := 100);
      ReactorLevel : FB_CTRL_PI(SET_POINT := 65, KP := 0.8, KI := 0.8, LIM_L := 0, LIM_H := 120);
      SeparatorTemp : FB_CTRL_PI(KP := -4, KI := -1, LIM_L := 0, LIM_H := 100);
      RectorTemperature : FB_CTRL_PI(SET_POINT := 122.9, KP := -8, KI := -1, LIM_L := 0, LIM_H := 100);
      SERVER_4_5_0 : SERVER_4_5(QI := TRUE, ID := localhost:61001);
      E_CYCLE_4 : E_CYCLE(DT := T#50ms);
      SERVER_3_5_2 : SERVER_3_5(QI := TRUE, ID := localhost:61002);
      SERVER_3_5_3 : SERVER_3_5(QI := TRUE, ID := localhost:61003);
      ProductionRateInit : Init_ConditionREALtype(InitialCondition := -0.4489);
      Init_ConditionREALtype_0 : Init_ConditionREALtype(InitialCondition := 0.6323);
      REAL2REAL : REAL2REAL(IN := 4.36871996);
      REAL2REAL_0 : REAL2REAL(IN := 100);
    END_FBS
    EVENT_CONNECTIONS
      ProductionSetpoint.CNF TO ProductionRate.REQ;
      F_MUL_2.CNF TO KxProdSetpoint.REQ;
      KxProdSetpoint.CNF TO Fp_.REQ;
      E_CYCLE_3.EO TO AandCControl.RSP;
      AandCControl.IND TO xmeas23.REQ;
      AandCControl.IND TO xmeas25.REQ;
      xmeas25.CNF TO yAC.REQ;
      F_MUL_4.CNF TO xmeas23_2.REQ;
      xmeas23_2.CNF TO yA.REQ;
      yAC.CNF TO yAC_.REQ;
      yAC_.CNF TO yA.REQ;
      yA.CNF TO yA_.REQ;
      AandCControl.INITO TO yAcontrol.INIT;
      yAcontrol.INITO TO yACcontrol.INIT;
      yA_.CNF TO yAcontrol.REQ;
      yAC_.CNF TO yACcontrol.REQ;
      yACcontrol.CNF TO F_SUB_0.REQ;
      F_SUB_0.CNF TO Loop15.REQ;
      Loop15.CNF TO F_ADD_4.REQ;
      yACcontrol.INITO TO Delay_With_InitConditionREALtype.INIT;
      F_ADD_4.CNF TO Delay_With_InitConditionREALtype.Start_and_REQ;
      Delay_With_InitConditionREALtype.CNF TO F_ADD_4.REQ;
      F_ADD_4.CNF TO r4.REQ;
      yAcontrol.CNF TO F_ADD_5.REQ;
      F_ADD_5.CNF TO r1.REQ;
      yAcontrol.INITO TO Delay_With_InitConditionREALtype_0.INIT;
      F_ADD_5.CNF TO Delay_With_InitConditionREALtype_0.Start_and_REQ;
      Delay_With_InitConditionREALtype_0.CNF TO F_ADD_5.REQ;
      TIME2TIME_2.CNF TO E_CYCLE_3.START;
      Fp_.CNF TO Fp.REQ;
      Fp.CNF TO AFeedRateSetpoint.REQ;
      r1.CNF TO TIME2TIME_2.REQ;
      r4.CNF TO TIME2TIME_2.REQ;
      AFeedRateSetpoint.CNF TO AFeedRate.REQ;
      CFeedRateSetpoint.CNF TO CFeedRate.REQ;
      Fp.CNF TO CFeedRateSetpoint.REQ;
      AFeedRate.INITO TO CFeedRate.INIT;
      ProductionRate.INITO TO AFeedRate.INIT;
      MoleGSetpoint.CNF TO GinProduct.REQ;
      MoleGSetpoint.CNF TO FeedforwardREAL.REQPctGsp;
      Fp_.CNF TO FeedforwardREAL.RECFp;
      FeedforwardREAL.CNFr2 TO DFeedRateSetpoint.REQ;
      FeedforwardREAL.CNFr3 TO EFeedRateSetpoint.REQ;
      Fp.CNF TO DFeedRateSetpoint.REQ;
      Fp.CNF TO EFeedRateSetpoint.REQ;
      DFeedRateSetpoint.CNF TO DFeedRate.REQ;
      EFeedRateSetpoint.CNF TO EFeedRate.REQ;
      CFeedRate.INITO TO DFeedRate.INIT;
      RectorPressure.INITO TO SeparatorLeel.INIT;
      SeparatorLeel.INITO TO StripperLevel.INIT;
      StripperLevel.INITO TO PurgeRate.INIT;
      PurgeRate.INITO TO SeparatorFlowRate.INIT;
      SeparatorFlowRate.INITO TO StripperFlowRate.INIT;
      Fp.CNF TO r5.REQ;
      Fp.CNF TO r7.REQ;
      Fp.CNF TO r6.REQ;
      r5.CNF TO PurgeRate.REQ;
      r6.CNF TO SeparatorFlowRate.REQ;
      r7.CNF TO StripperFlowRate.REQ;
      StripperLevel.CNF TO r7.REQ;
      SeparatorLeel.CNF TO r6.REQ;
      RectorPressure.CNF TO r5.REQ;
      ReactorLevel.CNF TO SeparatorTemp.REQ;
      EFeedRate.INITO TO ReactorLevel.INIT;
      ReactorLevel.INITO TO SeparatorTemp.INIT;
      SeparatorTemp.INITO TO RectorTemperature.INIT;
      AandCControl.INITO TO AandCControl.RSP;
      E_CYCLE_4.EO TO SERVER_4_5_0.RSP;
      CFeedRate.CNF TO E_CYCLE_4.START;
      DFeedRate.CNF TO E_CYCLE_4.START;
      PurgeRate.CNF TO E_CYCLE_4.START;
      SeparatorFlowRate.CNF TO E_CYCLE_4.START;
      StripperFlowRate.CNF TO E_CYCLE_4.START;
      SeparatorTemp.CNF TO E_CYCLE_4.START;
      RectorTemperature.CNF TO E_CYCLE_4.START;
      EFeedRate.CNF TO E_CYCLE_4.START;
      E_CYCLE_4.EO TO SERVER_3_5_3.RSP;
      E_CYCLE_4.EO TO SERVER_3_5_2.RSP;
      SERVER_3_5_2.INITO TO SERVER_3_5_2.RSP;
      SERVER_3_5_3.INITO TO SERVER_3_5_3.RSP;
      SERVER_3_5_2.IND TO RectorPressure.REQ;
      SERVER_3_5_2.INITO TO RectorPressure.INIT;
      SERVER_3_5_3.INITO TO EFeedRate.INIT;
      SERVER_3_5_2.IND TO PurgeRate.REQ;
      SERVER_3_5_2.INITO TO SeparatorLeel.REQ;
      SERVER_3_5_2.IND TO SeparatorFlowRate.REQ;
      SERVER_3_5_2.IND TO StripperLevel.REQ;
      SERVER_3_5_3.IND TO StripperFlowRate.REQ;
      SERVER_3_5_3.IND TO ReactorLevel.REQ;
      SERVER_3_5_3.IND TO SeparatorTemp.REQ;
      SERVER_3_5_3.IND TO RectorTemperature.REQ;
      SERVER_3_5_3.IND TO EFeedRate.REQ;
      SERVER_4_5_0.IND TO ProductionSetpoint.REQ;
      SERVER_4_5_0.IND TO MoleGSetpoint.REQ;
      SERVER_4_5_0.IND TO AFeedRate.REQ;
      SERVER_4_5_0.IND TO CFeedRate.REQ;
      SERVER_4_5_0.IND TO DFeedRate.REQ;
      ProductionRate.INITO TO ProductionRateInit.InitEvent;
      ProductionRate.CNF TO ProductionRateInit.SubsequentEvent;
      ProductionRateInit.CNF TO Fp_.REQ;
      SERVER_4_5_0.INITO TO ProductionRate.INIT;
      SERVER_4_5_0.INITO TO GinProduct.INIT;
      SERVER_4_5_0.INITO TO SERVER_4_5_0.RSP;
      GinProduct.INITO TO Init_ConditionREALtype_0.InitEvent;
      GinProduct.CNF TO Init_ConditionREALtype_0.SubsequentEvent;
      Init_ConditionREALtype_0.CNF TO FeedforwardREAL.RECEadj;
      AFeedRate.CNF TO E_CYCLE_4.START;
      ProductionSetpoint.CNF TO REAL2REAL.REQ;
      REAL2REAL.CNF TO F_MUL_2.REQ;
      xmeas23.CNF TO REAL2REAL_0.REQ;
      REAL2REAL_0.CNF TO F_MUL_4.REQ;
    END_CONNECTIONS
    DATA_CONNECTIONS
      ProductionSetpoint.OUT TO ProductionRate.SET_POINT;
      ProductionSetpoint.OUT TO F_MUL_2.IN1;
      F_MUL_2.OUT TO KxProdSetpoint.IN;
      KxProdSetpoint.OUT TO Fp_.IN1;
      AandCControl.RD_1 TO xmeas23.IN;
      AandCControl.RD_2 TO xmeas25.IN;
      xmeas25.OUT TO yAC.IN2;
      xmeas23.OUT TO F_MUL_4.IN1;
      xmeas23.OUT TO yAC.IN1;
      F_MUL_4.OUT TO xmeas23_2.IN;
      xmeas23_2.OUT TO yA.IN1;
      yAC.OUT TO yAC_.IN;
      yAC_.OUT TO yA.IN2;
      yA.OUT TO yA_.IN;
      yA_.OUT TO yAcontrol.ACTUAL;
      yAC_.OUT TO yACcontrol.ACTUAL;
      yACcontrol.Y TO F_SUB_0.IN1;
      yAcontrol.Y TO F_SUB_0.IN2;
      F_SUB_0.OUT TO Loop15.IN;
      Loop15.OUT TO F_ADD_4.IN1;
      Delay_With_InitConditionREALtype.OUT TO F_ADD_4.IN2;
      F_ADD_4.OUT TO Delay_With_InitConditionREALtype.DelayedInput;
      F_ADD_4.OUT TO r4.IN;
      yAcontrol.Y TO F_ADD_5.IN1;
      F_ADD_5.OUT TO r1.IN;
      Delay_With_InitConditionREALtype_0.OUT TO F_ADD_5.IN2;
      F_ADD_5.OUT TO Delay_With_InitConditionREALtype_0.DelayedInput;
      TIME2TIME_2.OUT TO E_CYCLE_3.DT;
      Fp_.OUT TO Fp.IN;
      Fp.OUT TO AFeedRateSetpoint.IN1;
      r1.OUT TO AFeedRateSetpoint.IN2;
      AFeedRateSetpoint.OUT TO AFeedRate.SET_POINT;
      r4.OUT TO CFeedRateSetpoint.IN2;
      Fp.OUT TO CFeedRateSetpoint.IN1;
      CFeedRateSetpoint.OUT TO CFeedRate.SET_POINT;
      MoleGSetpoint.OUT TO GinProduct.SET_POINT;
      MoleGSetpoint.OUT TO FeedforwardREAL.PctGsp;
      Fp_.OUT TO FeedforwardREAL.Fp;
      FeedforwardREAL.r2 TO DFeedRateSetpoint.IN1;
      FeedforwardREAL.r3 TO EFeedRateSetpoint.IN1;
      Fp.OUT TO DFeedRateSetpoint.IN2;
      Fp.OUT TO EFeedRateSetpoint.IN2;
      DFeedRateSetpoint.OUT TO DFeedRate.SET_POINT;
      EFeedRateSetpoint.OUT TO EFeedRate.SET_POINT;
      Fp.OUT TO r5.IN1;
      Fp.OUT TO r6.IN1;
      Fp.OUT TO r7.IN1;
      RectorPressure.Y TO r5.IN2;
      SeparatorLeel.Y TO r6.IN2;
      StripperLevel.Y TO r7.IN2;
      r5.OUT TO PurgeRate.SET_POINT;
      r6.OUT TO SeparatorFlowRate.SET_POINT;
      r7.OUT TO StripperFlowRate.SET_POINT;
      ReactorLevel.Y TO SeparatorTemp.SET_POINT;
      SERVER_4_5_0.RD_1 TO ProductionRate.ACTUAL;
      SERVER_4_5_0.RD_2 TO GinProduct.ACTUAL;
      SERVER_4_5_0.RD_3 TO AFeedRate.ACTUAL;
      SERVER_4_5_0.RD_4 TO CFeedRate.ACTUAL;
      SERVER_4_5_0.RD_5 TO DFeedRate.ACTUAL;
      CFeedRate.Y TO SERVER_4_5_0.SD_2;
      DFeedRate.Y TO SERVER_4_5_0.SD_3;
      TIME2TIME_2.OUT TO Delay_With_InitConditionREALtype_0.DelayTime;
      TIME2TIME_2.OUT TO Delay_With_InitConditionREALtype.DelayTime;
      PurgeRate.Y TO SERVER_3_5_2.SD_1;
      SeparatorFlowRate.Y TO SERVER_3_5_2.SD_2;
      StripperFlowRate.Y TO SERVER_3_5_2.SD_3;
      SeparatorTemp.Y TO SERVER_3_5_3.SD_1;
      RectorTemperature.Y TO SERVER_3_5_3.SD_2;
      EFeedRate.Y TO SERVER_3_5_3.SD_3;
      SERVER_3_5_2.RD_1 TO RectorPressure.ACTUAL;
      SERVER_3_5_2.RD_2 TO PurgeRate.ACTUAL;
      SERVER_3_5_2.RD_3 TO SeparatorLeel.ACTUAL;
      SERVER_3_5_2.RD_4 TO SeparatorFlowRate.ACTUAL;
      SERVER_3_5_2.RD_5 TO StripperLevel.ACTUAL;
      SERVER_3_5_3.RD_1 TO StripperFlowRate.ACTUAL;
      SERVER_3_5_3.RD_2 TO ReactorLevel.ACTUAL;
      SERVER_3_5_3.RD_3 TO SeparatorTemp.ACTUAL;
      SERVER_3_5_3.RD_4 TO RectorTemperature.ACTUAL;
      SERVER_3_5_3.RD_5 TO EFeedRate.ACTUAL;
      ProductionRate.Y TO ProductionRateInit.SubsequentInput;
      ProductionRateInit.OUT TO Fp_.IN2;
      ProductionRateInit.OUT TO SERVER_4_5_0.SD_4;
      Init_ConditionREALtype_0.OUT TO FeedforwardREAL.Eadj;
      GinProduct.Y TO Init_ConditionREALtype_0.SubsequentInput;
      AFeedRate.Y TO SERVER_4_5_0.SD_1;
      REAL2REAL.OUT TO F_MUL_2.IN2;
      REAL2REAL_0.OUT TO F_MUL_4.IN2;
    END_CONNECTIONS
  END_APPLICATION
  APPLICATION App1_ReactTempandSeptTemp
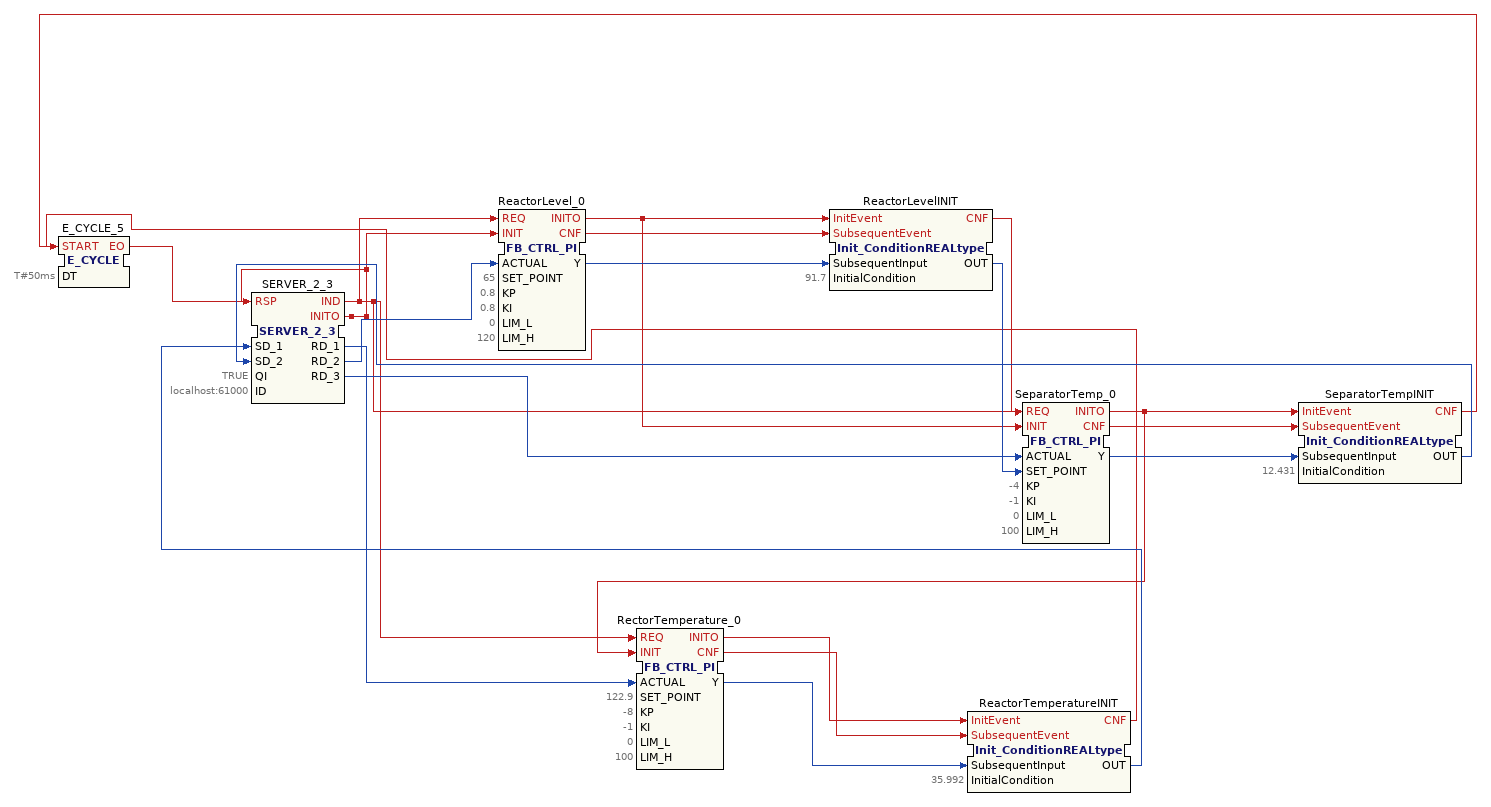
    FBS
      SeparatorTemp_0 : FB_CTRL_PI(KP := -4, KI := -1, LIM_L := 0, LIM_H := 100);
      ReactorLevel_0 : FB_CTRL_PI(SET_POINT := 65, KP := 0.8, KI := 0.8, LIM_L := 0, LIM_H := 120);
      RectorTemperature_0 : FB_CTRL_PI(SET_POINT := 122.9, KP := -8, KI := -1, LIM_L := 0, LIM_H := 100);
      E_CYCLE_5 : E_CYCLE(DT := T#50ms);
      SERVER_2_3 : SERVER_2_3(QI := TRUE, ID := localhost:61000);
      ReactorLevelINIT : Init_ConditionREALtype(InitialCondition := 91.7);
      SeparatorTempINIT : Init_ConditionREALtype(InitialCondition := 12.431);
      ReactorTemperatureINIT : Init_ConditionREALtype(InitialCondition := 35.992);
    END_FBS
    EVENT_CONNECTIONS
      SERVER_2_3.IND TO ReactorLevel_0.REQ;
      SERVER_2_3.INITO TO ReactorLevel_0.INIT;
      SERVER_2_3.IND TO SeparatorTemp_0.REQ;
      SERVER_2_3.IND TO RectorTemperature_0.REQ;
      E_CYCLE_5.EO TO SERVER_2_3.RSP;
      ReactorLevel_0.INITO TO ReactorLevelINIT.InitEvent;
      ReactorLevel_0.INITO TO SeparatorTemp_0.INIT;
      ReactorLevel_0.CNF TO ReactorLevelINIT.SubsequentEvent;
      ReactorLevelINIT.CNF TO SeparatorTemp_0.REQ;
      SeparatorTemp_0.INITO TO SeparatorTempINIT.InitEvent;
      SeparatorTemp_0.INITO TO RectorTemperature_0.INIT;
      SeparatorTemp_0.CNF TO SeparatorTempINIT.SubsequentEvent;
      SeparatorTempINIT.CNF TO E_CYCLE_5.START;
      RectorTemperature_0.INITO TO ReactorTemperatureINIT.InitEvent;
      RectorTemperature_0.CNF TO ReactorTemperatureINIT.SubsequentEvent;
      ReactorTemperatureINIT.CNF TO E_CYCLE_5.START;
      SERVER_2_3.INITO TO SERVER_2_3.RSP;
    END_CONNECTIONS
    DATA_CONNECTIONS
      ReactorLevel_0.Y TO ReactorLevelINIT.SubsequentInput;
      SeparatorTemp_0.Y TO SeparatorTempINIT.SubsequentInput;
      RectorTemperature_0.Y TO ReactorTemperatureINIT.SubsequentInput;
      ReactorTemperatureINIT.OUT TO SERVER_2_3.SD_1;
      SeparatorTempINIT.OUT TO SERVER_2_3.SD_2;
      SERVER_2_3.RD_1 TO RectorTemperature_0.ACTUAL;
      SERVER_2_3.RD_2 TO ReactorLevel_0.ACTUAL;
      SERVER_2_3.RD_3 TO SeparatorTemp_0.ACTUAL;
      ReactorLevelINIT.OUT TO SeparatorTemp_0.SET_POINT;
    END_CONNECTIONS
  END_APPLICATION
  APPLICATION App2_SepLiquidLevel_and_FlowRate
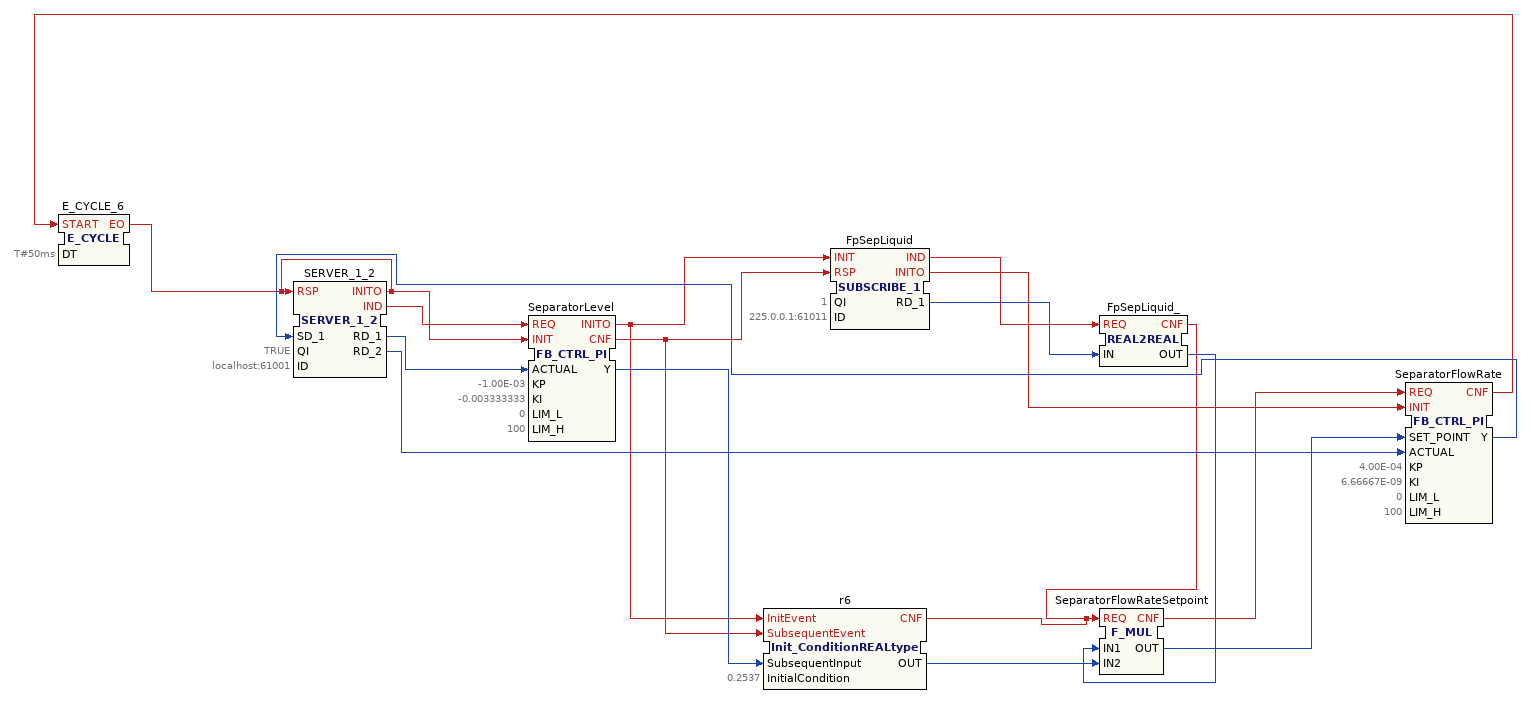
    FBS
      SeparatorLevel : FB_CTRL_PI(KP := -1.00E-03, KI := -0.003333333, LIM_L := 0, LIM_H := 100);
      r6 : Init_ConditionREALtype(InitialCondition := 0.2537);
      E_CYCLE_6 : E_CYCLE(DT := T#50ms);
      SERVER_1_2 : SERVER_1_2(QI := TRUE, ID := localhost:61001);
      FpSepLiquid : SUBSCRIBE_1(QI := 1, ID := 225.0.0.1:61011);
      SeparatorFlowRateSetpoint : F_MUL;
      FpSepLiquid_ : REAL2REAL;
      SeparatorFlowRate : FB_CTRL_PI(KP := 4.00E-04, KI := 6.66667E-09, LIM_L := 0, LIM_H := 100);
    END_FBS
    EVENT_CONNECTIONS
      SeparatorLevel.INITO TO r6.InitEvent;
      E_CYCLE_6.EO TO SERVER_1_2.RSP;
      SERVER_1_2.INITO TO SERVER_1_2.RSP;
      SERVER_1_2.IND TO SeparatorLevel.REQ;
      SERVER_1_2.INITO TO SeparatorLevel.INIT;
      SeparatorLevel.CNF TO r6.SubsequentEvent;
      SeparatorLevel.INITO TO FpSepLiquid.INIT;
      SeparatorLevel.CNF TO FpSepLiquid.RSP;
      FpSepLiquid.IND TO FpSepLiquid_.REQ;
      FpSepLiquid_.CNF TO SeparatorFlowRateSetpoint.REQ;
      r6.CNF TO SeparatorFlowRateSetpoint.REQ;
      SeparatorFlowRateSetpoint.CNF TO SeparatorFlowRate.REQ;
      FpSepLiquid.INITO TO SeparatorFlowRate.INIT;
      SeparatorFlowRate.CNF TO E_CYCLE_6.START;
    END_CONNECTIONS
    DATA_CONNECTIONS
      SeparatorLevel.Y TO r6.SubsequentInput;
      FpSepLiquid.RD_1 TO FpSepLiquid_.IN;
      FpSepLiquid_.OUT TO SeparatorFlowRateSetpoint.IN1;
      r6.OUT TO SeparatorFlowRateSetpoint.IN2;
      SERVER_1_2.RD_1 TO SeparatorLevel.ACTUAL;
      SeparatorFlowRateSetpoint.OUT TO SeparatorFlowRate.SET_POINT;
      SERVER_1_2.RD_2 TO SeparatorFlowRate.ACTUAL;
      SeparatorFlowRate.Y TO SERVER_1_2.SD_1;
    END_CONNECTIONS
  END_APPLICATION
  APPLICATION App3_StripperLiquidLevel_and_FlowRate
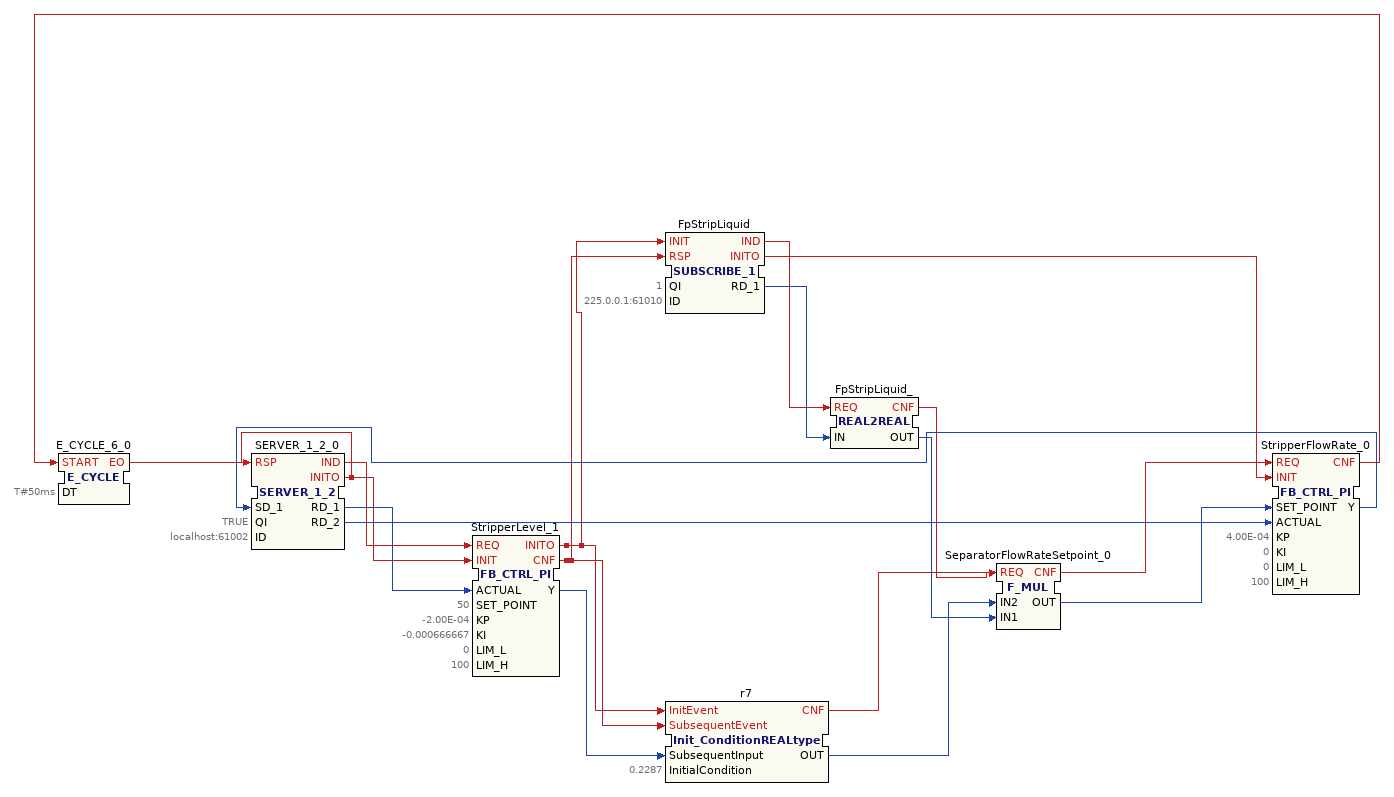
    FBS
      StripperLevel_1 : FB_CTRL_PI(SET_POINT := 50, KP := -2.00E-04, KI := -0.000666667, LIM_L := 0, LIM_H := 100);
      StripperFlowRate_0 : FB_CTRL_PI(KP := 4.00E-04, KI := 0, LIM_L := 0, LIM_H := 100);
      SERVER_1_2_0 : SERVER_1_2(QI := TRUE, ID := localhost:61002);
      E_CYCLE_6_0 : E_CYCLE(DT := T#50ms);
      FpStripLiquid : SUBSCRIBE_1(QI := 1, ID := 225.0.0.1:61010);
      FpStripLiquid_ : REAL2REAL;
      r7 : Init_ConditionREALtype(InitialCondition := 0.2287);
      SeparatorFlowRateSetpoint_0 : F_MUL;
    END_FBS
    EVENT_CONNECTIONS
      E_CYCLE_6_0.EO TO SERVER_1_2_0.RSP;
      SERVER_1_2_0.IND TO StripperLevel_1.REQ;
      SERVER_1_2_0.INITO TO StripperLevel_1.INIT;
      StripperLevel_1.INITO TO r7.InitEvent;
      StripperLevel_1.CNF TO r7.SubsequentEvent;
      r7.CNF TO SeparatorFlowRateSetpoint_0.REQ;
      StripperLevel_1.INITO TO FpStripLiquid.INIT;
      StripperLevel_1.CNF TO FpStripLiquid.RSP;
      FpStripLiquid.IND TO FpStripLiquid_.REQ;
      FpStripLiquid_.CNF TO SeparatorFlowRateSetpoint_0.REQ;
      SeparatorFlowRateSetpoint_0.CNF TO StripperFlowRate_0.REQ;
      FpStripLiquid.INITO TO StripperFlowRate_0.INIT;
      SERVER_1_2_0.INITO TO SERVER_1_2_0.RSP;
      StripperFlowRate_0.CNF TO E_CYCLE_6_0.START;
    END_CONNECTIONS
    DATA_CONNECTIONS
      StripperLevel_1.Y TO r7.SubsequentInput;
      r7.OUT TO SeparatorFlowRateSetpoint_0.IN2;
      FpStripLiquid_.OUT TO SeparatorFlowRateSetpoint_0.IN1;
      FpStripLiquid.RD_1 TO FpStripLiquid_.IN;
      SeparatorFlowRateSetpoint_0.OUT TO StripperFlowRate_0.SET_POINT;
      StripperFlowRate_0.Y TO SERVER_1_2_0.SD_1;
      SERVER_1_2_0.RD_1 TO StripperLevel_1.ACTUAL;
      SERVER_1_2_0.RD_2 TO StripperFlowRate_0.ACTUAL;
    END_CONNECTIONS
  END_APPLICATION
  APPLICATION App4_PressureControl
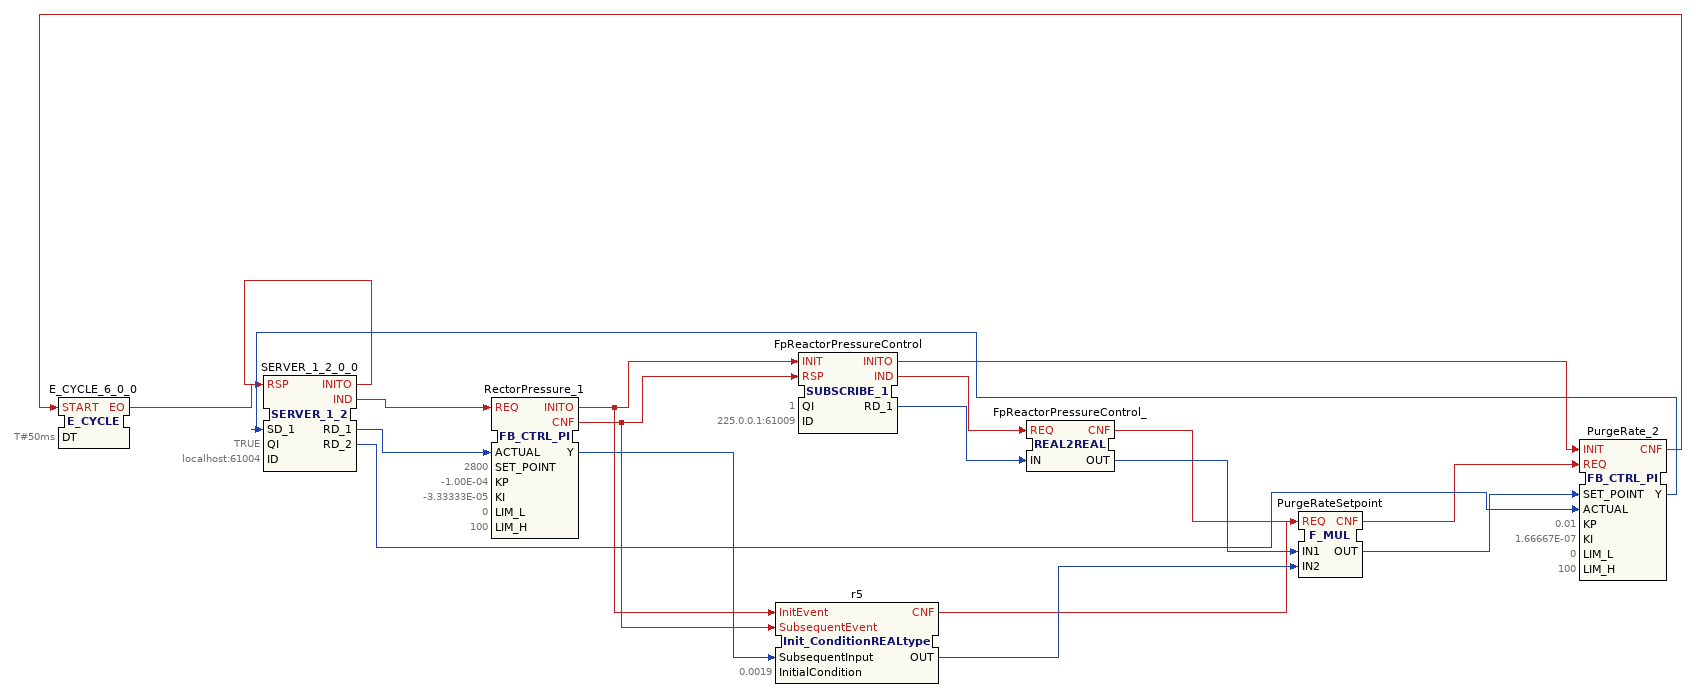
    FBS
      RectorPressure_1 : FB_CTRL_PI(SET_POINT := 2800, KP := -1.00E-04, KI := -3.33333E-05, LIM_L := 0, LIM_H := 100);
      PurgeRate_2 : FB_CTRL_PI(KP := 0.01, KI := 1.66667E-07, LIM_L := 0, LIM_H := 100);
      E_CYCLE_6_0_0 : E_CYCLE(DT := T#50ms);
      SERVER_1_2_0_0 : SERVER_1_2(QI := TRUE, ID := localhost:61004);
      r5 : Init_ConditionREALtype(InitialCondition := 0.0019);
      FpReactorPressureControl : SUBSCRIBE_1(QI := 1, ID := 225.0.0.1:61009);
      FpReactorPressureControl_ : REAL2REAL;
      PurgeRateSetpoint : F_MUL;
    END_FBS
    EVENT_CONNECTIONS
      SERVER_1_2_0_0.INITO TO SERVER_1_2_0_0.RSP;
      E_CYCLE_6_0_0.EO TO SERVER_1_2_0_0.RSP;
      SERVER_1_2_0_0.IND TO RectorPressure_1.REQ;
      RectorPressure_1.INITO TO r5.InitEvent;
      RectorPressure_1.CNF TO r5.SubsequentEvent;
      RectorPressure_1.INITO TO FpReactorPressureControl.INIT;
      FpReactorPressureControl.INITO TO PurgeRate_2.INIT;
      RectorPressure_1.CNF TO FpReactorPressureControl.RSP;
      FpReactorPressureControl.IND TO FpReactorPressureControl_.REQ;
      FpReactorPressureControl_.CNF TO PurgeRateSetpoint.REQ;
      r5.CNF TO PurgeRateSetpoint.REQ;
      PurgeRateSetpoint.CNF TO PurgeRate_2.REQ;
      PurgeRate_2.CNF TO E_CYCLE_6_0_0.START;
    END_CONNECTIONS
    DATA_CONNECTIONS
      FpReactorPressureControl.RD_1 TO FpReactorPressureControl_.IN;
      FpReactorPressureControl_.OUT TO PurgeRateSetpoint.IN1;
      r5.OUT TO PurgeRateSetpoint.IN2;
      PurgeRateSetpoint.OUT TO PurgeRate_2.SET_POINT;
      PurgeRate_2.Y TO SERVER_1_2_0_0.SD_1;
      SERVER_1_2_0_0.RD_1 TO RectorPressure_1.ACTUAL;
      SERVER_1_2_0_0.RD_2 TO PurgeRate_2.ACTUAL;
      RectorPressure_1.Y TO r5.SubsequentInput;
    END_CONNECTIONS
  END_APPLICATION
  APPLICATION App5_ProductionRateandQualityControl
    FBS
      TIME2TIME_2_0 : TIME2TIME(IN := T#100ms);
      E_CYCLE_4_0 : E_CYCLE(DT := T#50ms);
      E_CYCLE_3_0 : E_CYCLE;
      ProductionRateFbt : ProductionRateFbt(INITCOND := -0.4489, SET_POINT_Xmeas17 := 22.89, KP := 3.2, KI := 6.4, LIM_L := -30, LIM_H := 30);
      SERVER_2_0 : SERVER_2(QI := TRUE, ID := localhost:61005);
      AandCReactants : AandCReactants(SETPOINT_yAcontrol := 63.137, KP_yAcontrol := 2.00E-04, KI_yAcontrol := 0.0002, SET_POINT_yACcontrol := 51, KP_yACcontrol := 3.00E-04, KI_yACcontrol := 0.0006, InitialCondition_r1 := 0.002722836244293, InitialCondition_r4 := 0.092236609900323, INITCOND_AFeedRate := 26.248, KP_AFeedRate := 0.001, KI_AFeedRate := 0, LIM_L_AFeedRate := 0, LIM_H_AFeedRate := 100, INITCOND_CFeedRate := 60.566, KP_CFeedRate := 0.003, KI_CFeedRate := 0.00000005, LIM_L_CFeedRate := 0, LIM_H_CFeedRate := 100);
      PercentGinProduct : PercentGinProduct(INITCOND_Eadj := 0.6323, KP_PercentGinProduct := -0.4, KI_PercentGinProduct := -0.666666667, LIM_L_PercentGinProduct := -1000000000000, LIM_H_PercentGinProduct := 1000000000000, INITCOND_XMV1 := 62.807, KP_DFeedRate := 1.60E-06, KI_DFeedRate := 0, LIM_L_DFeedRate := 0, LIM_H_DFeedRate := 100, INITCOND_XMV2 := 53.2867, KP_EFeedRate := 1.80E-06, KI_EFeedRate := 0, LIM_L_EFeedRate := 0, LIM_H_FeedRate := 100);
      REAL2REAL_1 : REAL2REAL;
      SERVER_0_2 : SERVER_0_2(QI := TRUE, ID := localhost:61006);
      SERVER_3_5_4 : SERVER_3_5(QI := TRUE, ID := localhost:61007);
      PUBLISH_1 : PUBLISH_1;
      PUBLISH_1_0 : PUBLISH_1(QI := 1, ID := 225.0.0.1:61008);
    END_FBS
    EVENT_CONNECTIONS
      TIME2TIME_2_0.CNF TO E_CYCLE_3_0.START;
      SERVER_2_0.INITO TO SERVER_2_0.RSP;
      E_CYCLE_3_0.EO TO SERVER_2_0.RSP;
      SERVER_2_0.INITO TO AandCReactants.INIT_yACandYAcontrol;
      SERVER_2_0.IND TO AandCReactants.REQ_yACandYAcontrol;
      AandCReactants.CNF TO TIME2TIME_2_0.REQ;
      ProductionRateFbt.INITO TO PercentGinProduct.INIT;
      SERVER_3_5_4.INITO TO ProductionRateFbt.INIT;
      SERVER_3_5_4.IND TO REAL2REAL_1.REQ;
      SERVER_3_5_4.IND TO ProductionRateFbt.REQ;
      ProductionRateFbt.CNF TO PercentGinProduct.REQ;
      SERVER_3_5_4.IND TO PercentGinProduct.REQ;
      PercentGinProduct.CNF TO E_CYCLE_4_0.START;
      E_CYCLE_4_0.EO TO SERVER_0_2.RSP;
      E_CYCLE_4_0.EO TO SERVER_3_5_4.RSP;
      SERVER_0_2.INITO TO SERVER_3_5_4.INIT;
      SERVER_3_5_4.INITO TO SERVER_3_5_4.RSP;
      SERVER_0_2.INITO TO SERVER_0_2.RSP;
      PercentGinProduct.INITO TO PUBLISH_1.INIT;
      ProductionRateFbt.CNF TO PUBLISH_1.REQ;
      PUBLISH_1.CNF TO E_CYCLE_4_0.START;
      ProductionRateFbt.CNF TO PUBLISH_1_0.REQ;
      ProductionRateFbt.INITO TO PUBLISH_1_0.INIT;
    END_CONNECTIONS
    DATA_CONNECTIONS
      TIME2TIME_2_0.OUT TO E_CYCLE_3_0.DT;
      SERVER_2_0.RD_1 TO AandCReactants.XMEAS23;
      SERVER_2_0.RD_2 TO AandCReactants.XMEAS25;
      AandCReactants.XMV3 TO SERVER_2_0.SD_1;
      AandCReactants.XMV4 TO SERVER_2_0.SD_2;
      ProductionRateFbt.Fp TO PercentGinProduct.Fp;
      SERVER_0_2.RD_1 TO AandCReactants.ACTUAL_AFeedRate_Xmeas1;
      SERVER_0_2.RD_2 TO AandCReactants.ACTUAL_CFeedRate_Xmeas4;
      PercentGinProduct.XMV1 TO SERVER_3_5_4.SD_1;
      PercentGinProduct.XMV2 TO SERVER_3_5_4.SD_2;
      ProductionRateFbt.PRODSP TO SERVER_3_5_4.SD_3;
      SERVER_3_5_4.RD_1 TO ProductionRateFbt.ACT_Xmeas17;
      SERVER_3_5_4.RD_2 TO PercentGinProduct.ACT_PercentGinProduct_Xmeas40;
      SERVER_3_5_4.RD_3 TO PercentGinProduct.ACT_DFeedRate_Xmeas2;
      SERVER_3_5_4.RD_4 TO PercentGinProduct.ACT_E_FeedRate_Xmeas3;
      SERVER_3_5_4.RD_5 TO REAL2REAL_1.IN;
      TIME2TIME_2_0.OUT TO AandCReactants.DelaySampleTime_yACandYAcontrol;
      ProductionRateFbt.Fp TO AandCReactants.Fp;
      ProductionRateFbt.Fp TO PUBLISH_1.SD_1;
      ProductionRateFbt.Fp TO PUBLISH_1_0.SD_1;
    END_CONNECTIONS
  END_APPLICATION
  DEVICE FORTE_PC_1 : FORTE_PC(MGR_ID := "localhost:61499")
    {SET_ATTRIBUTE(Profile, HOLOBLOC)}
    RESOURCE EMB_RES : EMB_RES
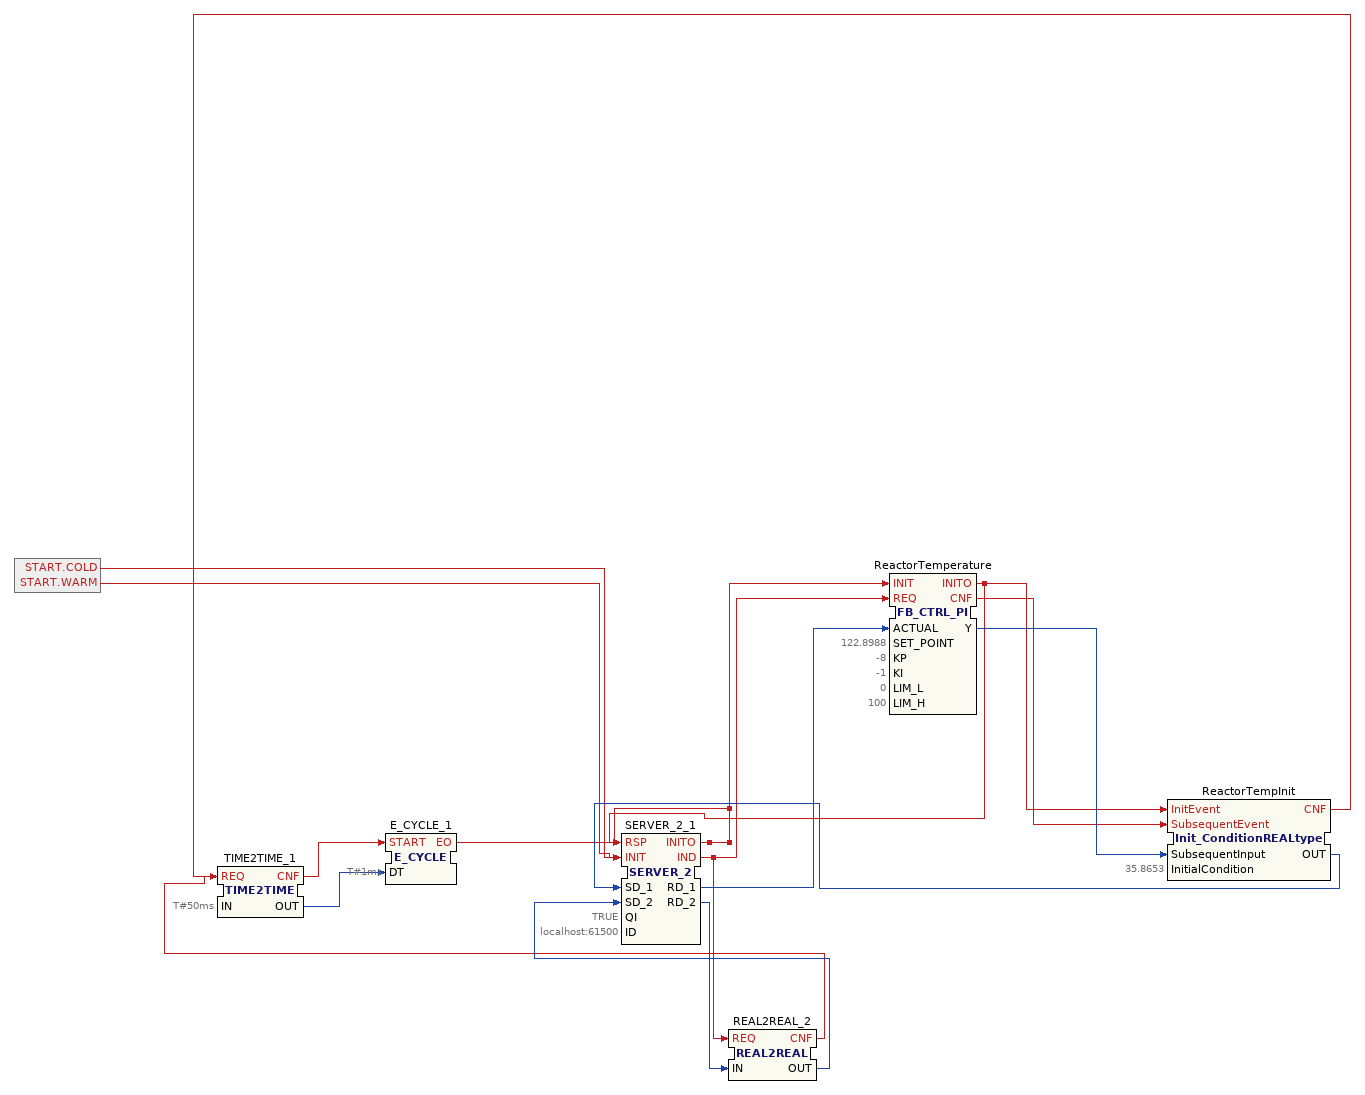
      FBS
        TIME2TIME_1 : TIME2TIME(IN := T#50ms);
        E_CYCLE_1 : E_CYCLE(DT := T#1ms);
        SERVER_2_1 : SERVER_2(QI := TRUE, ID := localhost:61500);
        ReactorTemperature : FB_CTRL_PI(SET_POINT := 122.8988, KP := -8, KI := -1, LIM_L := 0, LIM_H := 100);
        ReactorTempInit : Init_ConditionREALtype(InitialCondition := 35.8653);
        REAL2REAL_2 : REAL2REAL;
      END_FBS
      EVENT_CONNECTIONS
        TIME2TIME_1.CNF TO E_CYCLE_1.START;
        E_CYCLE_1.EO TO SERVER_2_1.RSP;
        SERVER_2_1.INITO TO ReactorTemperature.INIT;
        SERVER_2_1.IND TO ReactorTemperature.REQ;
        ReactorTemperature.INITO TO SERVER_2_1.RSP;
        ReactorTemperature.INITO TO ReactorTempInit.InitEvent;
        ReactorTemperature.CNF TO ReactorTempInit.SubsequentEvent;
        ReactorTempInit.CNF TO TIME2TIME_1.REQ;
        START.COLD TO SERVER_2_1.INIT;
        START.WARM TO SERVER_2_1.INIT;
        SERVER_2_1.IND TO REAL2REAL_2.REQ;
        REAL2REAL_2.CNF TO TIME2TIME_1.REQ;
        SERVER_2_1.INITO TO SERVER_2_1.RSP;
      END_CONNECTIONS
      DATA_CONNECTIONS
        TIME2TIME_1.OUT TO E_CYCLE_1.DT;
        SERVER_2_1.RD_1 TO ReactorTemperature.ACTUAL;
        ReactorTemperature.Y TO ReactorTempInit.SubsequentInput;
        ReactorTempInit.OUT TO SERVER_2_1.SD_1;
        SERVER_2_1.RD_2 TO REAL2REAL_2.IN;
        REAL2REAL_2.OUT TO SERVER_2_1.SD_2;
      END_CONNECTIONS
    END_RESOURCE
  END_DEVICE
  MAPPINGS
    reactortemperatureloop.TIME2TIME_1 ON FORTE_PC_1.EMB_RES.TIME2TIME_1;
    reactortemperatureloop.E_CYCLE_1 ON FORTE_PC_1.EMB_RES.E_CYCLE_1;
    reactortemperatureloop.SERVER_2_1 ON FORTE_PC_1.EMB_RES.SERVER_2_1;
    reactortemperatureloop.ReactorTemperature ON FORTE_PC_1.EMB_RES.ReactorTemperature;
    reactortemperatureloop.ReactorTempInit ON FORTE_PC_1.EMB_RES.ReactorTempInit;
    reactortemperatureloop.REAL2REAL_2 ON FORTE_PC_1.EMB_RES.REAL2REAL_2;
  END_MAPPINGS
  SEGMENTS
    Ethernet : Ethernet;
  END_SEGMENTS
  LINKS
    FORTE_PC_1 => Ethernet;
  END_LINKS
END_SYSTEM
